C05374=1023.242,179.277,-116.475,168.477,48.773,159.154
C05375=1023.248,179.526,-116.498,168.481,48.767,159.153
C05376=1023.253,179.776,-116.521,168.485,48.762,159.153
C05377=1023.259,180.025,-116.544,168.489,48.757,159.152
C05378=1023.265,180.273,-116.565,168.492,48.752,159.151
C05379=1023.270,180.522,-116.588,168.496,48.746,159.151
C05380=1023.276,180.771,-116.611,168.501,48.741,159.151
C05381=1023.282,181.020,-116.632,168.504,48.735,159.150
C05382=1023.288,181.269,-116.655,168.508,48.730,159.149
C05383=1023.294,181.518,-116.678,168.511,48.725,159.149
C05384=1023.299,181.767,-116.701,168.516,48.719,159.148
C05385=1023.305,182.015,-116.723,168.519,48.714,159.148
C05386=1023.311,182.264,-116.745,168.523,48.708,159.147
C05387=1023.317,182.513,-116.768,168.526,48.703,159.147
C05388=1023.322,182.762,-116.791,168.531,48.698,159.146
C05389=1023.327,183.012,-116.814,168.534,48.693,159.146
C05390=1023.333,183.261,-116.837,168.537,48.688,159.145
C05391=1023.338,183.510,-116.861,168.541,48.683,159.145
C05392=1023.343,183.759,-116.884,168.545,48.678,159.144
C05393=1023.349,184.007,-116.906,168.549,48.673,159.144
C05394=1023.354,184.256,-116.930,168.553,48.668,159.143
C05395=1023.359,184.505,-116.953,168.556,48.662,159.143
C05396=1023.365,184.754,-116.976,168.560,48.657,159.142
C05397=1023.370,185.003,-117.000,168.564,48.652,159.142
C05398=1023.376,185.251,-117.023,168.568,48.647,159.141
C05399=1023.382,185.500,-117.046,168.571,48.642,159.141
C05400=1023.386,185.749,-117.069,168.575,48.637,159.140
C05401=1023.392,185.998,-117.092,168.579,48.632,159.140
C05402=1023.398,186.247,-117.115,168.582,48.627,159.139
C05403=1023.403,186.496,-117.138,168.587,48.622,159.139
C05404=1023.408,186.745,-117.161,168.590,48.616,159.138
C05405=1023.414,186.994,-117.184,168.594,48.611,159.138
C05406=1023.419,187.243,-117.208,168.598,48.606,159.137
C05407=1023.425,187.525,-117.234,168.603,48.600,159.137
C05408=1023.432,187.806,-117.261,168.607,48.594,159.136
C05409=1023.438,188.088,-117.287,168.611,48.589,159.136
C05410=1023.445,188.371,-117.313,168.615,48.583,159.135
C05411=1023.450,188.620,-117.337,168.619,48.578,159.135
C05412=1023.456,188.869,-117.360,168.623,48.573,159.134
C05413=1023.461,189.117,-117.383,168.627,48.568,159.134
C05414=1023.466,189.366,-117.406,168.631,48.563,159.133
C05415=1023.472,189.614,-117.430,168.635,48.558,159.133
C05416=1023.477,189.864,-117.453,168.638,48.552,159.132
C05417=1023.482,190.113,-117.476,168.643,48.547,159.132
C05418=1023.488,190.361,-117.499,168.646,48.542,159.131
C05419=1023.494,190.610,-117.524,168.651,48.537,159.131
C05420=1023.499,190.859,-117.547,168.654,48.532,159.130
C05421=1023.505,191.108,-117.570,168.658,48.527,159.130
C05422=1023.511,191.358,-117.593,168.662,48.521,159.129
C05423=1023.517,191.606,-117.617,168.666,48.517,159.129
C05424=1023.522,191.855,-117.640,168.670,48.512,159.128
C05425=1023.527,192.104,-117.664,168.674,48.507,159.128
C05426=1023.533,192.352,-117.687,168.678,48.502,159.127
C05427=1023.538,192.602,-117.711,168.681,48.496,159.127
C05428=1023.544,192.850,-117.734,168.686,48.491,159.126
C05429=1023.550,193.099,-117.757,168.690,48.486,159.126
C05430=1023.555,193.348,-117.781,168.694,48.481,159.125
C05431=1023.561,193.596,-117.805,168.698,48.476,159.125
C05432=1023.567,193.845,-117.828,168.701,48.471,159.125
C05433=1023.572,194.094,-117.851,168.706,48.465,159.124
C05434=1023.578,194.343,-117.875,168.710,48.460,159.124
C05435=1023.583,194.592,-117.898,168.713,48.456,159.123
C05436=1023.590,194.841,-117.922,168.718,48.450,159.123
C05437=1023.595,195.090,-117.945,168.721,48.446,159.122
C05438=1023.601,195.338,-117.970,168.726,48.440,159.122
C05439=1023.606,195.587,-117.992,168.730,48.435,159.121
C05440=1023.612,195.835,-118.016,168.733,48.430,159.121
C05441=1023.617,196.085,-118.040,168.738,48.425,159.120
C05442=1023.624,196.334,-118.064,168.742,48.420,159.120
C05443=1023.629,196.583,-118.087,168.746,48.415,159.119
C05444=1023.635,196.831,-118.111,168.750,48.410,159.119
C05445=1023.641,197.080,-118.134,168.754,48.405,159.119
C05446=1023.646,197.329,-118.158,168.758,48.400,159.118
C05447=1023.652,197.578,-118.181,168.762,48.395,159.118
C05448=1023.658,197.827,-118.206,168.766,48.389,159.117
C05449=1023.664,198.075,-118.229,168.770,48.384,159.117
C05450=1023.669,198.324,-118.252,168.774,48.379,159.116
C05451=1023.675,198.573,-118.277,168.779,48.374,159.116
C05452=1023.681,198.822,-118.300,168.782,48.369,159.115
C05453=1023.686,199.071,-118.324,168.787,48.364,159.115
C05454=1023.692,199.319,-118.348,168.791,48.359,159.114
C05455=1023.698,199.568,-118.371,168.795,48.354,159.114
C05456=1023.704,199.817,-118.395,168.799,48.349,159.113
C05457=1023.709,200.066,-118.420,168.803,48.344,159.113
C05458=1023.715,200.314,-118.443,168.807,48.339,159.113
C05459=1023.720,200.563,-118.467,168.811,48.334,159.112
C05460=1023.726,200.813,-118.491,168.816,48.329,159.112
C05461=1023.732,201.061,-118.516,168.819,48.324,159.111
C05462=1023.738,201.309,-118.539,168.824,48.319,159.111
C05463=1023.743,201.558,-118.564,168.828,48.314,159.110
C05464=1023.749,201.807,-118.588,168.832,48.309,159.110
C05465=1023.754,202.056,-118.612,168.836,48.304,159.109
C05466=1023.760,202.305,-118.635,168.841,48.300,159.109
C05467=1023.765,202.553,-118.660,168.844,48.295,159.109
C05468=1023.771,202.803,-118.684,168.849,48.290,159.108
C05469=1023.776,203.051,-118.709,168.853,48.285,159.108
C05470=1023.782,203.300,-118.732,168.857,48.280,159.107
C05471=1023.805,204.331,-118.833,169.270,48.380,159.187
C05472=1023.816,204.745,-118.876,169.275,48.373,159.186
C05473=1023.827,205.160,-118.919,169.281,48.366,159.186
C05474=1023.838,205.574,-118.961,169.286,48.359,159.185
C05475=1023.849,205.988,-119.004,169.292,48.352,159.184
C05476=1023.856,206.237,-119.031,169.295,48.349,159.184
C05477=1023.862,206.486,-119.056,169.298,48.344,159.184
C05478=1023.868,206.734,-119.082,169.301,48.341,159.183
C05479=1023.874,206.982,-119.108,169.305,48.336,159.183
C05480=1023.882,207.231,-119.134,169.307,48.333,159.182
C05481=1023.888,207.480,-119.159,169.311,48.329,159.182
C05482=1023.894,207.728,-119.185,169.314,48.325,159.182
C05483=1023.900,207.976,-119.211,169.318,48.321,159.181
C05484=1023.908,208.225,-119.237,169.320,48.317,159.181
C05485=1023.913,208.474,-119.263,169.324,48.313,159.180
C05486=1023.920,208.722,-119.289,169.327,48.309,159.180
C05487=1023.926,208.972,-119.315,169.331,48.305,159.180
C05488=1023.933,209.220,-119.341,169.333,48.301,159.179
C05489=1023.939,209.468,-119.367,169.337,48.297,159.179
C05490=1023.946,209.717,-119.393,169.340,48.293,159.179
C05491=1023.952,209.965,-119.419,169.344,48.289,159.178
C05492=1023.958,210.214,-119.445,169.346,48.285,159.178
C05493=1023.965,210.462,-119.471,169.350,48.282,159.178
C05494=1023.972,210.711,-119.497,169.353,48.278,159.177
C05495=1023.978,210.959,-119.524,169.356,48.274,159.177
C05496=1023.984,211.208,-119.549,169.360,48.270,159.176
C05497=1023.991,211.457,-119.575,169.362,48.266,159.176
C05498=1023.997,211.705,-119.602,169.366,48.263,159.176
C05499=1024.003,211.954,-119.627,169.369,48.259,159.175
C05500=1024.009,212.203,-119.654,169.373,48.255,159.175
C05501=1024.016,212.451,-119.681,169.376,48.251,159.175
C05502=1024.022,212.699,-119.707,169.379,48.247,159.174
C05503=1024.029,212.948,-119.734,169.382,48.244,159.174
C05504=1024.035,213.197,-119.759,169.386,48.240,159.174
C05505=1024.042,213.445,-119.785,169.389,48.236,159.173
C05506=1024.048,213.694,-119.812,169.393,48.232,159.173
C05507=1024.054,213.942,-119.838,169.396,48.229,159.173
C05508=1024.061,214.191,-119.865,169.399,48.225,159.172
C05509=1024.067,214.439,-119.890,169.402,48.221,159.172
C05510=1024.073,214.688,-119.916,169.406,48.217,159.172
C05511=1024.080,214.937,-119.943,169.409,48.214,159.171
C05512=1024.086,215.185,-119.970,169.412,48.210,159.171
C05513=1024.093,215.433,-119.996,169.415,48.206,159.171
C05514=1024.099,215.682,-120.023,169.418,48.202,159.170
C05515=1024.106,215.930,-120.049,169.422,48.198,159.170
C05516=1024.112,216.179,-120.076,169.425,48.195,159.170
C05517=1024.119,216.427,-120.102,169.429,48.191,159.169
C05518=1024.125,216.676,-120.127,169.432,48.187,159.169
C05519=1024.131,216.925,-120.154,169.435,48.183,159.169
C05520=1024.138,217.173,-120.181,169.439,48.180,159.168
C05521=1024.145,217.421,-120.207,169.442,48.176,159.168
C05522=1024.151,217.670,-120.234,169.445,48.172,159.168
C05523=1024.158,217.919,-120.260,169.449,48.169,159.167
C05524=1024.164,218.168,-120.287,169.452,48.165,159.167
C05525=1024.171,218.416,-120.313,169.456,48.161,159.167
C05526=1024.178,218.664,-120.339,169.459,48.158,159.166
C05527=1024.183,218.913,-120.366,169.462,48.154,159.166
C05528=1024.194,219.329,-120.410,169.468,48.148,159.165
C05529=1024.205,219.746,-120.456,169.474,48.142,159.165
C05530=1024.215,220.162,-120.500,169.479,48.136,159.165
C05531=1024.227,220.579,-120.545,169.485,48.130,159.164
C05532=1024.232,220.828,-120.572,169.488,48.127,159.164
C05533=1024.239,221.077,-120.599,169.491,48.123,159.163
C05534=1024.245,221.325,-120.625,169.495,48.120,159.163
C05535=1024.252,221.574,-120.652,169.498,48.116,159.163
C05536=1024.258,221.822,-120.679,169.502,48.112,159.163
C05537=1024.265,222.070,-120.706,169.505,48.109,159.162
C05538=1024.271,222.319,-120.732,169.509,48.105,159.162
C05539=1024.277,222.568,-120.759,169.512,48.102,159.162
C05540=1024.284,222.815,-120.786,169.516,48.098,159.161
C05541=1024.290,223.064,-120.813,169.519,48.095,159.161
C05542=1024.297,223.313,-120.840,169.521,48.091,159.161
C05543=1024.303,223.561,-120.866,169.525,48.088,159.161
C05544=1024.310,223.810,-120.894,169.529,48.085,159.160
C05545=1024.316,224.058,-120.921,169.532,48.080,159.160
C05546=1024.323,224.307,-120.947,169.535,48.077,159.160
C05547=1024.329,224.555,-120.975,169.539,48.074,159.160
C05548=1024.335,224.804,-121.002,169.542,48.070,159.159
C05549=1024.342,225.053,-121.028,169.546,48.067,159.159
C05550=1024.348,225.300,-121.055,169.549,48.064,159.159
C05551=1024.355,225.549,-121.082,169.553,48.060,159.158
C05552=1024.361,225.797,-121.108,169.556,48.056,159.158
C05553=1024.368,226.046,-121.136,169.560,48.053,159.158
C05554=1024.374,226.295,-121.163,169.563,48.049,159.158
C05555=1024.380,226.543,-121.190,169.567,48.046,159.157
C05556=1024.388,226.791,-121.217,169.570,48.043,159.157
C05557=1024.394,227.040,-121.244,169.573,48.039,159.157
C05558=1024.400,227.288,-121.271,169.577,48.035,159.157
C05559=1024.406,227.537,-121.298,169.580,48.032,159.156
C05560=1024.412,227.785,-121.326,169.584,48.029,159.156
C05561=1024.420,228.034,-121.352,169.587,48.026,159.156
C05562=1024.426,228.282,-121.380,169.591,48.022,159.156
C05563=1024.432,228.531,-121.406,169.594,48.019,159.155
C05564=1024.439,228.779,-121.434,169.598,48.015,159.155
C05565=1024.445,229.028,-121.461,169.601,48.012,159.155
C05566=1024.451,229.276,-121.489,169.604,48.009,159.155
C05567=1024.458,229.524,-121.516,169.608,48.006,159.154
C05568=1024.464,229.773,-121.543,169.611,48.003,159.154
C05569=1024.470,230.021,-121.571,169.616,47.999,159.154
C05570=1024.477,230.269,-121.598,169.618,47.995,159.154
C05571=1024.483,230.519,-121.625,169.622,47.992,159.153
C05572=1024.490,230.767,-121.653,169.625,47.989,159.153
C05573=1024.496,231.015,-121.681,169.629,47.986,159.153
C05574=1024.502,231.264,-121.708,169.633,47.982,159.153
C05575=1024.509,231.512,-121.735,169.636,47.979,159.153
C05576=1024.515,231.760,-121.763,169.640,47.976,159.152
C05577=1024.522,232.009,-121.790,169.643,47.973,159.152
C05578=1024.528,232.257,-121.817,169.647,47.969,159.152
C05579=1024.534,232.505,-121.845,169.650,47.966,159.152
C05580=1024.541,232.754,-121.872,169.653,47.963,159.151
C05581=1024.548,233.002,-121.900,169.657,47.960,159.151
C05582=1024.553,233.251,-121.928,169.660,47.957,159.151
C05583=1024.559,233.499,-121.955,169.664,47.953,159.151
C05584=1024.570,233.908,-122.000,169.670,47.949,159.151
C05585=1024.581,234.317,-122.045,169.676,47.943,159.150
C05586=1024.591,234.726,-122.092,169.682,47.938,159.150
C05587=1024.602,235.134,-122.137,169.688,47.932,159.150
C05588=1024.609,235.383,-122.165,169.691,47.929,159.149
C05589=1024.615,235.631,-122.192,169.695,47.926,159.149
C05590=1024.622,235.880,-122.219,169.698,47.923,159.149
C05591=1024.628,236.129,-122.247,169.702,47.919,159.149
C05592=1024.634,236.377,-122.274,169.705,47.917,159.149
C05593=1024.641,236.625,-122.302,169.709,47.914,159.148
C05594=1024.647,236.874,-122.331,169.712,47.910,159.148
C05595=1024.654,237.122,-122.358,169.717,47.907,159.148
C05596=1024.660,237.371,-122.386,169.720,47.904,159.148
C05597=1024.667,237.619,-122.414,169.723,47.901,159.147
C05598=1024.673,237.867,-122.441,169.727,47.898,159.148
C05599=1024.680,238.115,-122.469,169.730,47.895,159.147
C05600=1024.686,238.364,-122.497,169.734,47.892,159.147
C05601=1024.693,238.612,-122.525,169.737,47.888,159.147
C05602=1024.699,238.861,-122.553,169.741,47.885,159.147
C05603=1024.706,239.109,-122.580,169.745,47.883,159.147
C05604=1024.713,239.358,-122.608,169.749,47.879,159.146
C05605=1024.719,239.606,-122.636,169.752,47.876,159.146
C05606=1024.725,239.854,-122.664,169.755,47.873,159.146
C05607=1024.732,240.102,-122.692,169.759,47.870,159.146
C05608=1024.738,240.351,-122.720,169.763,47.867,159.146
C05609=1024.744,240.599,-122.748,169.767,47.864,159.145
C05610=1024.751,240.848,-122.776,169.770,47.861,159.145
C05611=1024.757,241.096,-122.805,169.774,47.858,159.145
C05612=1024.764,241.344,-122.833,169.777,47.855,159.145
C05613=1024.770,241.593,-122.861,169.781,47.852,159.145
C05614=1024.776,241.841,-122.888,169.785,47.849,159.145
C05615=1024.783,242.089,-122.917,169.788,47.847,159.145
C05616=1024.789,242.337,-122.945,169.792,47.843,159.144
C05617=1024.795,242.586,-122.973,169.795,47.840,159.144
C05618=1024.802,242.834,-123.002,169.800,47.837,159.144
C05619=1024.808,243.082,-123.030,169.803,47.834,159.144
C05620=1024.814,243.331,-123.058,169.806,47.832,159.144
C05621=1024.821,243.579,-123.086,169.810,47.829,159.144
C05622=1024.828,243.827,-123.114,169.814,47.826,159.144
C05623=1024.834,244.076,-123.143,169.818,47.823,159.143
C05624=1024.840,244.324,-123.172,169.821,47.820,159.143
C05625=1024.847,244.573,-123.199,169.824,47.817,159.143
C05626=1024.853,244.821,-123.228,169.829,47.814,159.143
C05627=1024.859,245.070,-123.257,169.832,47.812,159.143
C05628=1024.865,245.317,-123.285,169.836,47.809,159.143
C05629=1024.871,245.565,-123.313,169.840,47.806,159.143
C05630=1024.878,245.814,-123.342,169.843,47.803,159.143
C05631=1024.884,246.062,-123.371,169.847,47.800,159.143
C05632=1024.891,246.310,-123.399,169.850,47.798,159.143
C05633=1024.897,246.558,-123.428,169.855,47.795,159.142
C05634=1024.903,246.807,-123.456,169.858,47.792,159.142
C05635=1024.909,247.055,-123.485,169.861,47.790,159.142
C05636=1024.916,247.304,-123.513,169.865,47.786,159.142
C05637=1024.922,247.552,-123.542,169.869,47.784,159.142
C05638=1024.928,247.800,-123.571,169.873,47.781,159.142
C05639=1024.935,248.048,-123.599,169.876,47.778,159.142
C05640=1024.945,248.451,-123.645,169.882,47.773,159.141
C05641=1024.955,248.854,-123.693,169.888,47.769,159.141
C05642=1024.966,249.256,-123.739,169.895,47.765,159.141
C05643=1024.976,249.660,-123.785,169.901,47.760,159.141
C05644=1024.983,249.908,-123.814,169.904,47.758,159.141
C05645=1024.990,250.156,-123.843,169.909,47.755,159.141
C05646=1024.996,250.404,-123.872,169.912,47.752,159.141
C05647=1025.002,250.652,-123.900,169.916,47.749,159.141
C05648=1025.009,250.900,-123.928,169.920,47.747,159.141
C05649=1025.015,251.148,-123.958,169.923,47.744,159.141
C05650=1025.021,251.397,-123.987,169.927,47.741,159.141
C05651=1025.027,251.645,-124.015,169.931,47.738,159.140
C05652=1025.035,251.894,-124.044,169.935,47.736,159.140
C05653=1025.041,252.142,-124.073,169.938,47.733,159.140
C05654=1025.047,252.390,-124.102,169.943,47.731,159.140
C05655=1025.053,252.638,-124.131,169.946,47.728,159.140
C05656=1025.060,252.887,-124.159,169.950,47.725,159.140
C05657=1025.066,253.135,-124.188,169.954,47.722,159.140
C05658=1025.073,253.383,-124.217,169.958,47.720,159.140
C05659=1025.080,253.631,-124.245,169.962,47.717,159.140
C05660=1025.086,253.880,-124.274,169.965,47.715,159.140
C05661=1025.093,254.128,-124.304,169.969,47.712,159.140
C05662=1025.099,254.376,-124.333,169.972,47.709,159.139
C05663=1025.106,254.624,-124.361,169.977,47.706,159.139
C05664=1025.113,254.872,-124.390,169.980,47.704,159.139
C05665=1025.119,255.121,-124.419,169.985,47.701,159.139
C05666=1025.125,255.369,-124.448,169.988,47.699,159.139
C05667=1025.132,255.617,-124.476,169.992,47.696,159.139
C05668=1025.139,255.866,-124.506,169.996,47.693,159.139
C05669=1025.145,256.114,-124.535,170.000,47.691,159.139
C05670=1025.151,256.362,-124.564,170.003,47.688,159.139
C05671=1025.158,256.610,-124.592,170.008,47.685,159.139
C05672=1025.165,256.859,-124.622,170.011,47.683,159.139
C05673=1025.171,257.107,-124.651,170.016,47.680,159.139
C05674=1025.178,257.355,-124.680,170.019,47.677,159.139
C05675=1025.186,257.603,-124.709,170.023,47.675,159.139
C05676=1025.192,257.851,-124.738,170.027,47.672,159.139
C05677=1025.198,258.099,-124.767,170.031,47.670,159.139
C05678=1025.204,258.347,-124.796,170.035,47.667,159.139
C05679=1025.212,258.596,-124.825,170.039,47.664,159.139
C05680=1025.218,258.844,-124.854,170.043,47.662,159.139
C05681=1025.224,259.092,-124.883,170.047,47.659,159.139
C05682=1025.231,259.341,-124.913,170.050,47.657,159.138
C05683=1025.238,259.589,-124.941,170.055,47.654,159.138
C05684=1025.245,259.838,-124.970,170.058,47.652,159.138
C05685=1025.252,260.085,-125.000,170.063,47.649,159.138
C05686=1025.258,260.333,-125.029,170.066,47.647,159.138
C05687=1025.266,260.582,-125.058,170.070,47.644,159.138
C05688=1025.272,260.830,-125.087,170.074,47.641,159.138
C05689=1025.278,261.078,-125.117,170.079,47.639,159.138
C05690=1025.284,261.327,-125.147,170.082,47.637,159.138
C05691=1025.291,261.575,-125.176,170.086,47.634,159.138
C05692=1025.297,261.822,-125.206,170.090,47.632,159.138
C05693=1025.304,262.071,-125.235,170.094,47.629,159.138
C05694=1025.311,262.319,-125.265,170.098,47.627,159.138
C05695=1025.317,262.567,-125.294,170.102,47.625,159.138
C05696=1025.327,262.968,-125.343,170.108,47.621,159.138
C05697=1025.338,263.369,-125.390,170.115,47.617,159.138
C05698=1025.348,263.771,-125.438,170.121,47.614,159.138
C05699=1025.359,264.172,-125.486,170.128,47.609,159.138
C05700=1025.365,264.420,-125.516,170.132,47.607,159.138
C05701=1025.372,264.668,-125.545,170.136,47.605,159.138
C05702=1025.379,264.916,-125.575,170.140,47.602,159.138
C05703=1025.384,265.164,-125.604,170.143,47.600,159.138
C05704=1025.391,265.413,-125.634,170.148,47.598,159.138
C05705=1025.398,265.660,-125.664,170.151,47.596,159.138
C05706=1025.405,265.909,-125.694,170.156,47.593,159.138
C05707=1025.411,266.156,-125.723,170.159,47.591,159.138
C05708=1025.418,266.405,-125.754,170.164,47.588,159.138
C05709=1025.424,266.653,-125.783,170.168,47.587,159.139
C05710=1025.431,266.901,-125.813,170.172,47.584,159.139
C05711=1025.437,267.149,-125.844,170.176,47.582,159.139
C05712=1025.444,267.398,-125.873,170.180,47.579,159.139
C05713=1025.450,267.645,-125.903,170.184,47.578,159.139
C05714=1025.458,267.894,-125.933,170.188,47.575,159.139
C05715=1025.463,268.141,-125.963,170.192,47.573,159.139
C05716=1025.470,268.390,-125.993,170.196,47.571,159.139
C05717=1025.476,268.638,-126.023,170.200,47.569,159.139
C05718=1025.483,268.886,-126.053,170.205,47.566,159.139
C05719=1025.490,269.134,-126.083,170.208,47.564,159.139
C05720=1025.496,269.382,-126.114,170.213,47.562,159.139
C05721=1025.503,269.630,-126.143,170.216,47.560,159.139
C05722=1025.510,269.879,-126.173,170.221,47.557,159.139
C05723=1025.515,270.126,-126.203,170.225,47.555,159.139
C05724=1025.523,270.375,-126.233,170.229,47.553,159.139
C05725=1025.528,270.623,-126.264,170.233,47.551,159.139
C05726=1025.536,270.871,-126.294,170.237,47.549,159.139
C05727=1025.541,271.119,-126.324,170.241,47.546,159.139
C05728=1025.549,271.367,-126.354,170.246,47.544,159.140
C05729=1025.555,271.615,-126.385,170.249,47.543,159.140
C05730=1025.562,271.863,-126.415,170.254,47.540,159.140
C05731=1025.568,272.111,-126.445,170.257,47.538,159.140
C05732=1025.575,272.359,-126.475,170.262,47.536,159.140
C05733=1025.581,272.607,-126.506,170.266,47.534,159.140
C05734=1025.588,272.856,-126.536,170.270,47.532,159.140
C05735=1025.594,273.103,-126.566,170.274,47.530,159.140
C05736=1025.601,273.352,-126.596,170.279,47.528,159.140
C05737=1025.607,273.599,-126.628,170.282,47.526,159.140
C05738=1025.614,273.847,-126.658,170.287,47.523,159.140
C05739=1025.621,274.096,-126.688,170.292,47.521,159.140
C05740=1025.627,274.343,-126.718,170.295,47.520,159.141
C05741=1025.634,274.592,-126.749,170.300,47.517,159.141
C05742=1025.640,274.840,-126.780,170.304,47.516,159.141
C05743=1025.647,275.087,-126.810,170.308,47.513,159.141
C05744=1025.653,275.336,-126.841,170.312,47.511,159.141
C05745=1025.661,275.584,-126.871,170.317,47.509,159.141
C05746=1025.666,275.832,-126.901,170.320,47.507,159.141
C05747=1025.673,276.079,-126.933,170.325,47.505,159.141
C05748=1025.680,276.328,-126.963,170.329,47.504,159.141
C05749=1025.687,276.576,-126.993,170.333,47.501,159.141
C05750=1025.693,276.824,-127.023,170.337,47.499,159.142
C05751=1025.700,277.072,-127.055,170.342,47.497,159.142
C05752=1025.711,277.478,-127.105,170.348,47.494,159.142
C05753=1025.721,277.883,-127.155,170.356,47.491,159.142
C05754=1025.732,278.289,-127.205,170.362,47.488,159.142
C05755=1025.743,278.695,-127.257,170.370,47.485,159.143
C05756=1025.749,278.943,-127.287,170.374,47.483,159.143
C05757=1025.756,279.190,-127.318,170.379,47.481,159.143
C05758=1025.762,279.439,-127.348,170.382,47.479,159.143
C05759=1025.769,279.687,-127.380,170.387,47.477,159.143
C05760=1025.776,279.935,-127.411,170.391,47.475,159.143
C05761=1025.782,280.182,-127.442,170.395,47.473,159.143
C05762=1025.788,280.431,-127.472,170.399,47.472,159.144
C05763=1025.795,280.679,-127.504,170.404,47.470,159.144
C05764=1025.802,280.926,-127.535,170.408,47.468,159.144
C05765=1025.809,281.175,-127.565,170.413,47.466,159.144
C05766=1025.815,281.422,-127.596,170.417,47.464,159.144
C05767=1025.821,281.671,-127.627,170.421,47.463,159.144
C05768=1025.828,281.919,-127.659,170.426,47.461,159.145
C05769=1025.835,282.167,-127.690,170.430,47.459,159.145
C05770=1025.842,282.415,-127.720,170.434,47.457,159.145
C05771=1025.849,282.663,-127.752,170.438,47.455,159.145
C05772=1025.855,282.911,-127.783,170.443,47.454,159.145
C05773=1025.861,283.158,-127.814,170.448,47.452,159.145
C05774=1025.868,283.406,-127.845,170.452,47.450,159.146
C05775=1025.875,283.654,-127.876,170.456,47.448,159.146
C05776=1025.881,283.902,-127.908,170.460,47.447,159.146
C05777=1025.889,284.150,-127.938,170.465,47.445,159.146
C05778=1025.895,284.398,-127.969,170.469,47.443,159.146
C05779=1025.902,284.646,-128.001,170.474,47.441,159.146
C05780=1025.909,284.894,-128.032,170.478,47.439,159.147
C05781=1025.915,285.142,-128.064,170.482,47.438,159.147
C05782=1025.922,285.390,-128.095,170.487,47.436,159.147
C05783=1025.929,285.638,-128.126,170.491,47.434,159.147
C05784=1025.935,285.886,-128.157,170.496,47.432,159.147
C05785=1025.941,286.133,-128.188,170.501,47.430,159.148
C05786=1025.948,286.381,-128.220,170.505,47.429,159.148
C05787=1025.955,286.629,-128.251,170.509,47.427,159.148
C05788=1025.962,286.877,-128.282,170.513,47.426,159.148
C05789=1025.968,287.125,-128.314,170.518,47.424,159.148
C05790=1025.975,287.373,-128.345,170.523,47.422,159.149
C05791=1025.982,287.621,-128.377,170.527,47.421,159.149
C05792=1025.989,287.868,-128.409,170.532,47.419,159.149
C05793=1025.995,288.116,-128.440,170.536,47.418,159.149
C05794=1026.001,288.364,-128.472,170.540,47.416,159.150
C05795=1026.008,288.612,-128.504,170.545,47.414,159.150
C05796=1026.015,288.860,-128.535,170.549,47.413,159.150
C05797=1026.022,289.108,-128.567,170.554,47.411,159.150
C05798=1026.028,289.356,-128.598,170.558,47.409,159.150
C05799=1026.035,289.603,-128.630,170.563,47.408,159.151
C05800=1026.043,289.852,-128.662,170.568,47.406,159.151
C05801=1026.049,290.100,-128.694,170.572,47.405,159.151
C05802=1026.055,290.348,-128.725,170.576,47.403,159.151
C05803=1026.062,290.596,-128.757,170.581,47.401,159.152
C05804=1026.069,290.843,-128.789,170.586,47.400,159.152
C05805=1026.076,291.091,-128.821,170.590,47.398,159.152
C05806=1026.082,291.339,-128.853,170.594,47.397,159.152
C05807=1026.089,291.586,-128.885,170.599,47.395,159.153
C05808=1026.101,292.005,-128.938,170.607,47.393,159.153
C05809=1026.112,292.423,-128.992,170.615,47.390,159.153
C05810=1026.123,292.840,-129.046,170.623,47.388,159.154
C05811=1026.134,293.259,-129.099,170.630,47.385,159.154
C05812=1026.141,293.506,-129.131,170.635,47.384,159.155
C05813=1026.148,293.755,-129.164,170.640,47.382,159.155
C05814=1026.155,294.002,-129.196,170.644,47.381,159.155
C05815=1026.161,294.250,-129.228,170.649,47.379,159.155
C05816=1026.168,294.498,-129.260,170.654,47.378,159.156
C05817=1026.174,294.745,-129.293,170.658,47.377,159.156
C05818=1026.180,294.993,-129.325,170.663,47.375,159.156
C05819=1026.187,295.241,-129.357,170.667,47.374,159.157
C05820=1026.194,295.489,-129.390,170.672,47.373,159.157
C05821=1026.201,295.736,-129.422,170.677,47.371,159.157
C05822=1026.207,295.985,-129.454,170.681,47.370,159.158
C05823=1026.213,296.232,-129.487,170.686,47.369,159.158
C05824=1026.221,296.479,-129.519,170.690,47.368,159.158
C05825=1026.227,296.728,-129.552,170.695,47.366,159.158
C05826=1026.233,296.976,-129.584,170.700,47.365,159.159
C05827=1026.240,297.223,-129.616,170.704,47.364,159.159
C05828=1026.247,297.471,-129.649,170.709,47.362,159.159
C05829=1026.253,297.718,-129.682,170.714,47.361,159.160
C05830=1026.261,297.966,-129.714,170.718,47.360,159.160
C05831=1026.267,298.215,-129.746,170.723,47.358,159.160
C05832=1026.273,298.462,-129.779,170.728,47.357,159.161
C05833=1026.280,298.709,-129.811,170.732,47.356,159.161
C05834=1026.287,298.958,-129.844,170.737,47.355,159.161
C05835=1026.294,299.205,-129.876,170.742,47.353,159.162
C05836=1026.300,299.453,-129.909,170.747,47.353,159.162
C05837=1026.307,299.701,-129.942,170.752,47.351,159.162
C05838=1026.314,299.948,-129.974,170.757,47.350,159.163
C05839=1026.320,300.196,-130.007,170.761,47.349,159.163
C05840=1026.327,300.444,-130.040,170.766,47.347,159.163
C05841=1026.334,300.691,-130.072,170.771,47.346,159.164
C05842=1026.341,300.939,-130.105,170.775,47.345,159.164
C05843=1026.347,301.187,-130.138,170.780,47.344,159.165
C05844=1026.355,301.435,-130.170,170.785,47.343,159.165
C05845=1026.361,301.683,-130.204,170.790,47.341,159.165
C05846=1026.368,301.930,-130.236,170.794,47.340,159.165
C05847=1026.375,302.178,-130.268,170.799,47.339,159.166
C05848=1026.382,302.426,-130.302,170.805,47.338,159.166
C05849=1026.388,302.673,-130.335,170.810,47.337,159.167
C05850=1026.396,302.921,-130.368,170.814,47.335,159.167
C05851=1026.402,303.169,-130.400,170.819,47.334,159.167
C05852=1026.408,303.416,-130.433,170.824,47.333,159.168
C05853=1026.416,303.664,-130.466,170.828,47.332,159.168
C05854=1026.422,303.912,-130.498,170.833,47.331,159.168
C05855=1026.430,304.159,-130.532,170.839,47.330,159.169
C05856=1026.437,304.407,-130.564,170.844,47.329,159.169
C05857=1026.444,304.655,-130.597,170.848,47.328,159.169
C05858=1026.450,304.903,-130.630,170.853,47.327,159.170
C05859=1026.458,305.150,-130.663,170.858,47.325,159.170
C05860=1026.464,305.397,-130.696,170.863,47.324,159.171
C05861=1026.471,305.646,-130.729,170.869,47.323,159.171
C05862=1026.479,305.893,-130.762,170.873,47.322,159.171
C05863=1026.485,306.141,-130.795,170.878,47.321,159.172
C05864=1026.491,306.358,-130.824,170.882,47.320,159.172
C05865=1026.497,306.576,-130.853,170.887,47.319,159.173
C05866=1026.504,306.794,-130.882,170.891,47.318,159.173
C05867=1026.510,307.012,-130.911,170.895,47.317,159.173
C05868=1026.516,307.228,-130.941,170.899,47.316,159.174
C05869=1026.522,307.446,-130.970,170.904,47.316,159.174
C05870=1026.529,307.664,-130.999,170.909,47.314,159.174
C05871=1026.534,307.882,-131.028,170.913,47.313,159.175
C05872=1026.542,308.130,-131.060,170.918,47.312,159.175
C05873=1026.548,308.377,-131.094,170.923,47.311,159.175
C05874=1026.555,308.625,-131.127,170.928,47.310,159.176
C05875=1026.563,308.873,-131.160,170.933,47.309,159.176
C05876=1026.570,309.120,-131.194,170.938,47.308,159.177
C05877=1026.577,309.368,-131.227,170.943,47.307,159.177
C05878=1026.584,309.616,-131.261,170.948,47.306,159.178
C05879=1026.591,309.863,-131.293,170.954,47.305,159.178
C05880=1026.598,310.110,-131.327,170.958,47.304,159.178
C05881=1026.605,310.358,-131.360,170.963,47.303,159.179
C05882=1026.612,310.605,-131.393,170.968,47.302,159.179
C05883=1026.620,310.853,-131.426,170.973,47.301,159.180
C05884=1026.626,311.101,-131.461,170.979,47.300,159.180
C05885=1026.633,311.348,-131.494,170.983,47.300,159.181
C05886=1026.640,311.596,-131.528,170.989,47.299,159.181
C05887=1026.647,311.843,-131.562,170.994,47.298,159.182
C05888=1026.653,312.091,-131.596,170.999,47.297,159.182
C05889=1026.660,312.338,-131.630,171.004,47.296,159.183
C05890=1026.667,312.586,-131.664,171.009,47.296,159.183
C05891=1026.674,312.834,-131.698,171.014,47.295,159.184
C05892=1026.680,313.081,-131.732,171.019,47.294,159.184
C05893=1026.688,313.329,-131.765,171.025,47.293,159.185
C05894=1026.694,313.577,-131.800,171.030,47.293,159.185
C05895=1026.701,313.824,-131.833,171.034,47.292,159.186
C05896=1026.708,314.071,-131.867,171.040,47.291,159.186
C05897=1026.714,314.319,-131.901,171.045,47.291,159.187
C05898=1026.721,314.567,-131.935,171.050,47.290,159.187
C05899=1026.729,314.815,-131.969,171.056,47.289,159.188
C05900=1026.735,315.062,-132.003,171.061,47.288,159.188
C05901=1026.742,315.309,-132.038,171.065,47.288,159.189
C05902=1026.749,315.557,-132.072,171.071,47.287,159.189
C05903=1026.756,315.805,-132.106,171.076,47.286,159.190
C05904=1026.763,316.052,-132.140,171.082,47.286,159.190
C05905=1026.770,316.300,-132.174,171.087,47.285,159.191
C05906=1026.776,316.547,-132.208,171.092,47.284,159.191
C05907=1026.783,316.794,-132.242,171.098,47.283,159.192
C05908=1026.791,317.042,-132.276,171.102,47.283,159.192
C05909=1026.797,317.290,-132.310,171.108,47.283,159.193
C05910=1026.805,317.537,-132.345,171.113,47.282,159.193
C05911=1026.812,317.785,-132.379,171.118,47.281,159.194
C05912=1026.818,318.033,-132.413,171.124,47.280,159.194
C05913=1026.826,318.280,-132.448,171.129,47.280,159.195
C05914=1026.833,318.527,-132.482,171.134,47.279,159.195
C05915=1026.840,318.775,-132.517,171.140,47.279,159.196
C05916=1026.847,319.022,-132.551,171.145,47.278,159.197
C05917=1026.854,319.270,-132.584,171.150,47.277,159.197
C05918=1026.861,319.517,-132.619,171.155,47.277,159.198
C05919=1026.868,319.765,-132.653,171.161,47.276,159.198
C05920=1026.876,320.012,-132.688,171.166,47.276,159.199
C05921=1026.882,320.260,-132.722,171.171,47.275,159.199
C05922=1026.890,320.507,-132.757,171.177,47.274,159.200
C05923=1026.897,320.755,-132.791,171.182,47.274,159.200
C05924=1026.903,320.975,-132.822,171.187,47.273,159.201
C05925=1026.909,321.196,-132.853,171.192,47.273,159.201
C05926=1026.915,321.415,-132.884,171.196,47.272,159.202
C05927=1026.922,321.636,-132.914,171.202,47.272,159.203
C05928=1026.928,321.856,-132.945,171.206,47.272,159.203
C05929=1026.935,322.076,-132.976,171.212,47.271,159.203
C05930=1026.941,322.296,-133.006,171.216,47.270,159.204
C05931=1026.948,322.516,-133.037,171.220,47.270,159.204
C05932=1026.955,322.763,-133.071,171.226,47.270,159.205
C05933=1026.962,323.011,-133.106,171.231,47.269,159.206
C05934=1026.970,323.258,-133.141,171.237,47.269,159.206
C05935=1026.977,323.506,-133.175,171.242,47.268,159.207
C05936=1026.984,323.754,-133.210,171.248,47.268,159.207
C05937=1026.991,324.001,-133.244,171.253,47.267,159.208
C05938=1026.999,324.248,-133.279,171.259,47.267,159.209
C05939=1027.006,324.496,-133.314,171.265,47.266,159.209
C05940=1027.013,324.743,-133.348,171.270,47.266,159.210
C05941=1027.020,324.991,-133.383,171.276,47.265,159.210
C05942=1027.028,325.239,-133.418,171.281,47.265,159.211
C05943=1027.036,325.486,-133.453,171.287,47.264,159.212
C05944=1027.042,325.733,-133.488,171.293,47.264,159.212
C05945=1027.050,325.981,-133.522,171.299,47.263,159.213
C05946=1027.057,326.229,-133.557,171.304,47.263,159.214
C05947=1027.064,326.476,-133.592,171.310,47.263,159.214
C05948=1027.073,326.723,-133.627,171.315,47.262,159.215
C05949=1027.079,326.971,-133.662,171.321,47.262,159.215
C05950=1027.087,327.218,-133.696,171.327,47.262,159.216
C05951=1027.094,327.466,-133.732,171.332,47.261,159.217
C05952=1027.102,327.713,-133.766,171.338,47.261,159.217
C05953=1027.109,327.960,-133.802,171.343,47.261,159.218
C05954=1027.116,328.208,-133.838,171.349,47.260,159.219
C05955=1027.123,328.455,-133.873,171.355,47.260,159.219
C05956=1027.130,328.703,-133.908,171.360,47.259,159.220
C05957=1027.138,328.950,-133.944,171.366,47.259,159.221
C05958=1027.145,329.197,-133.979,171.371,47.259,159.221
C05959=1027.152,329.444,-134.014,171.377,47.259,159.222
C05960=1027.159,329.692,-134.050,171.382,47.259,159.223
C05961=1027.166,329.939,-134.085,171.388,47.259,159.223
C05962=1027.173,330.187,-134.121,171.394,47.259,159.224
C05963=1027.181,330.434,-134.156,171.400,47.258,159.225
C05964=1027.188,330.681,-134.191,171.406,47.258,159.226
C05965=1027.195,330.929,-134.227,171.412,47.258,159.226
C05966=1027.202,331.176,-134.263,171.417,47.258,159.227
C05967=1027.210,331.424,-134.298,171.423,47.257,159.228
C05968=1027.217,331.671,-134.334,171.429,47.257,159.228
C05969=1027.225,331.918,-134.369,171.434,47.257,159.229
C05970=1027.232,332.165,-134.405,171.440,47.257,159.230
C05971=1027.239,332.413,-134.440,171.446,47.257,159.230
C05972=1027.247,332.660,-134.476,171.451,47.257,159.231
C05973=1027.254,332.908,-134.512,171.458,47.256,159.232
C05974=1027.262,333.156,-134.548,171.464,47.257,159.233
C05975=1027.269,333.402,-134.583,171.470,47.257,159.233
C05976=1027.277,333.650,-134.619,171.475,47.256,159.234
C05977=1027.284,333.897,-134.654,171.481,47.256,159.235
C05978=1027.292,334.144,-134.691,171.487,47.256,159.236
C05979=1027.298,334.392,-134.726,171.493,47.256,159.236
C05980=1027.306,334.639,-134.762,171.499,47.256,159.237
C05981=1027.313,334.887,-134.799,171.505,47.256,159.238
C05982=1027.320,335.134,-134.835,171.511,47.256,159.239
C05983=1027.328,335.381,-134.871,171.517,47.256,159.239
C05984=1027.334,335.598,-134.902,171.521,47.256,159.240
C05985=1027.340,335.817,-134.934,171.527,47.256,159.241
C05986=1027.348,336.035,-134.966,171.533,47.256,159.241
C05987=1027.354,336.252,-134.997,171.537,47.256,159.242
C05988=1027.360,336.470,-135.029,171.543,47.256,159.243
C05989=1027.367,336.688,-135.061,171.548,47.257,159.244
C05990=1027.373,336.906,-135.093,171.553,47.256,159.244
C05991=1027.380,337.124,-135.125,171.558,47.257,159.245
C05992=1027.387,337.372,-135.161,171.565,47.256,159.246
C05993=1027.394,337.618,-135.197,171.571,47.257,159.247
C05994=1027.402,337.866,-135.233,171.576,47.256,159.247
C05995=1027.410,338.113,-135.269,171.582,47.257,159.248
C05996=1027.417,338.361,-135.306,171.588,47.257,159.249
C05997=1027.424,338.608,-135.342,171.595,47.257,159.250
C05998=1027.432,338.855,-135.378,171.601,47.257,159.250
C05999=1027.439,339.102,-135.415,171.607,47.257,159.251
C06000=1027.447,339.349,-135.451,171.613,47.258,159.252
C06001=1027.455,339.597,-135.488,171.619,47.257,159.253
C06002=1027.462,339.844,-135.523,171.625,47.258,159.254
C06003=1027.470,340.091,-135.560,171.631,47.258,159.255
C06004=1027.478,340.338,-135.597,171.637,47.258,159.255
C06005=1027.485,340.586,-135.633,171.644,47.258,159.256
C06006=1027.492,340.833,-135.670,171.650,47.258,159.257
C06007=1027.500,341.080,-135.707,171.655,47.258,159.258
C06008=1027.507,341.328,-135.743,171.661,47.259,159.259
C06009=1027.514,341.574,-135.780,171.668,47.259,159.260
C06010=1027.522,341.821,-135.816,171.674,47.259,159.261
C06011=1027.529,342.068,-135.854,171.680,47.260,159.261
C06012=1027.537,342.316,-135.890,171.686,47.260,159.262
C06013=1027.544,342.563,-135.927,171.693,47.260,159.263
C06014=1027.552,342.810,-135.964,171.699,47.260,159.264
C06015=1027.560,343.057,-136.001,171.705,47.261,159.265
C06016=1027.567,343.305,-136.037,171.712,47.261,159.266
C06017=1027.575,343.552,-136.074,171.718,47.261,159.267
C06018=1027.583,343.799,-136.111,171.724,47.262,159.268
C06019=1027.590,344.046,-136.148,171.731,47.262,159.268
C06020=1027.598,344.293,-136.185,171.737,47.262,159.269
C06021=1027.605,344.540,-136.223,171.743,47.263,159.270
C06022=1027.613,344.788,-136.259,171.750,47.263,159.271
C06023=1027.620,345.035,-136.296,171.756,47.263,159.272
C06024=1027.628,345.282,-136.333,171.762,47.264,159.273
C06025=1027.635,345.529,-136.371,171.769,47.264,159.274
C06026=1027.643,345.776,-136.407,171.775,47.264,159.275
C06027=1027.651,346.023,-136.444,171.781,47.265,159.276
C06028=1027.658,346.270,-136.481,171.788,47.266,159.277
C06029=1027.667,346.518,-136.519,171.794,47.266,159.278
C06030=1027.674,346.765,-136.556,171.801,47.266,159.279
C06031=1027.682,347.012,-136.593,171.807,47.267,159.279
C06032=1027.689,347.259,-136.631,171.813,47.267,159.280
C06033=1027.697,347.506,-136.668,171.820,47.268,159.281
C06034=1027.704,347.753,-136.705,171.826,47.268,159.282
C06035=1027.712,348.000,-136.742,171.833,47.268,159.283
C06036=1027.720,348.247,-136.780,171.839,47.269,159.284
C06037=1027.728,348.494,-136.817,171.845,47.270,159.285
C06038=1027.735,348.741,-136.854,171.852,47.270,159.286
C06039=1027.743,348.989,-136.892,171.859,47.271,159.287
C06040=1027.751,349.235,-136.929,171.866,47.271,159.288
C06041=1027.759,349.483,-136.967,171.872,47.272,159.289
C06042=1027.766,349.730,-137.005,171.878,47.273,159.290
C06043=1027.774,349.977,-137.042,171.885,47.273,159.291
C06044=1027.781,350.193,-137.075,171.891,47.274,159.292
C06045=1027.787,350.409,-137.108,171.896,47.275,159.293
C06046=1027.795,350.626,-137.141,171.902,47.275,159.294
C06047=1027.801,350.842,-137.174,171.908,47.275,159.295
C06048=1027.808,351.058,-137.207,171.914,47.276,159.296
C06049=1027.815,351.275,-137.241,171.920,47.276,159.296
C06050=1027.821,351.491,-137.274,171.925,47.277,159.297
C06051=1027.828,351.707,-137.307,171.931,47.277,159.298
C06052=1027.836,351.954,-137.345,171.938,47.278,159.299
C06053=1027.844,352.201,-137.382,171.944,47.279,159.300
C06054=1027.851,352.448,-137.420,171.951,47.279,159.301
C06055=1027.859,352.695,-137.458,171.958,47.280,159.302
C06056=1027.867,352.942,-137.496,171.965,47.281,159.303
C06057=1027.876,353.190,-137.534,171.971,47.282,159.304
C06058=1027.883,353.436,-137.572,171.978,47.282,159.305
C06059=1027.890,353.683,-137.610,171.985,47.283,159.307
C06060=1027.898,353.930,-137.648,171.992,47.284,159.308
C06061=1027.907,354.177,-137.686,171.999,47.284,159.309
C06062=1027.915,354.424,-137.724,172.005,47.285,159.310
C06063=1027.922,354.671,-137.762,172.012,47.286,159.311
C06064=1027.931,354.918,-137.800,172.019,47.287,159.312
C06065=1027.938,355.165,-137.837,172.026,47.288,159.313
C06066=1027.946,355.412,-137.876,172.032,47.289,159.314
C06067=1027.954,355.659,-137.914,172.040,47.290,159.315
C06068=1027.962,355.906,-137.953,172.047,47.290,159.316
C06069=1027.970,356.152,-137.991,172.053,47.291,159.317
C06070=1027.978,356.400,-138.030,172.060,47.292,159.319
C06071=1027.986,356.647,-138.068,172.067,47.293,159.320
C06072=1027.994,356.893,-138.107,172.074,47.294,159.321
C06073=1028.002,357.141,-138.145,172.081,47.295,159.322
C06074=1028.009,357.387,-138.184,172.088,47.296,159.323
C06075=1028.017,357.634,-138.222,172.095,47.296,159.324
C06076=1028.026,357.882,-138.261,172.102,47.297,159.325
C06077=1028.033,358.128,-138.299,172.108,47.298,159.326
C06078=1028.042,358.375,-138.337,172.116,47.299,159.328
C06079=1028.050,358.622,-138.376,172.123,47.300,159.329
C06080=1028.058,358.868,-138.415,172.130,47.301,159.330
C06081=1028.066,359.115,-138.453,172.137,47.302,159.331
C06082=1028.074,359.362,-138.492,172.144,47.303,159.332
C06083=1028.082,359.609,-138.530,172.151,47.304,159.333
C06084=1028.090,359.856,-138.569,172.158,47.305,159.334
C06085=1028.098,360.103,-138.608,172.165,47.306,159.336
C06086=1028.107,360.350,-138.647,172.172,47.307,159.337
C06087=1028.115,360.597,-138.686,172.179,47.308,159.338
C06088=1028.122,360.843,-138.725,172.187,47.309,159.339
C06089=1028.130,361.090,-138.764,172.194,47.310,159.340
C06090=1028.139,361.337,-138.803,172.201,47.312,159.342
C06091=1028.147,361.584,-138.842,172.208,47.312,159.343
C06092=1028.154,361.831,-138.881,172.216,47.314,159.344
C06093=1028.162,362.077,-138.920,172.222,47.315,159.345
C06094=1028.170,362.324,-138.959,172.230,47.316,159.346
C06095=1028.179,362.571,-138.998,172.237,47.317,159.348
C06096=1028.187,362.818,-139.038,172.244,47.318,159.349
C06097=1028.195,363.065,-139.077,172.252,47.319,159.350
C06098=1028.203,363.311,-139.116,172.258,47.320,159.351
C06099=1028.210,363.558,-139.155,172.266,47.322,159.353
C06100=1028.219,363.805,-139.195,172.274,47.323,159.354
C06101=1028.227,364.052,-139.233,172.281,47.324,159.355
C06102=1028.235,364.298,-139.273,172.288,47.325,159.356
C06103=1028.243,364.545,-139.313,172.295,47.327,159.358
C06104=1028.251,364.765,-139.348,172.302,47.327,159.359
C06105=1028.258,364.984,-139.382,172.309,47.329,159.360
C06106=1028.266,365.204,-139.418,172.315,47.330,159.361
C06107=1028.272,365.424,-139.453,172.322,47.331,159.362
C06108=1028.280,365.643,-139.488,172.328,47.332,159.363
C06109=1028.288,365.862,-139.523,172.335,47.333,159.365
C06110=1028.295,366.082,-139.558,172.342,47.334,159.366
C06111=1028.302,366.302,-139.594,172.348,47.336,159.367
C06112=1028.311,366.549,-139.633,172.356,47.337,159.368
C06113=1028.319,366.795,-139.672,172.363,47.338,159.369
C06114=1028.327,367.042,-139.712,172.371,47.339,159.371
C06115=1028.336,367.289,-139.752,172.379,47.341,159.372
C06116=1028.344,367.535,-139.791,172.386,47.343,159.373
C06117=1028.352,367.782,-139.832,172.394,47.344,159.375
C06118=1028.360,368.028,-139.871,172.402,47.345,159.376
C06119=1028.370,368.276,-139.911,172.409,47.346,159.377
C06120=1028.378,368.522,-139.950,172.416,47.348,159.379
C06121=1028.386,368.768,-139.991,172.424,47.349,159.380
C06122=1028.394,369.015,-140.030,172.431,47.351,159.381
C06123=1028.402,369.262,-140.070,172.439,47.353,159.383
C06124=1028.412,369.509,-140.110,172.447,47.354,159.384
C06125=1028.419,369.755,-140.150,172.454,47.355,159.385
C06126=1028.427,370.002,-140.191,172.462,47.357,159.387
C06127=1028.436,370.248,-140.230,172.470,47.358,159.388
C06128=1028.444,370.495,-140.271,172.477,47.360,159.390
C06129=1028.453,370.741,-140.311,172.485,47.362,159.391
C06130=1028.461,370.988,-140.351,172.493,47.363,159.392
C06131=1028.469,371.235,-140.392,172.501,47.365,159.394
C06132=1028.478,371.481,-140.432,172.509,47.366,159.395
C06133=1028.486,371.728,-140.472,172.516,47.368,159.397
C06134=1028.495,371.974,-140.512,172.524,47.369,159.398
C06135=1028.503,372.221,-140.553,172.533,47.371,159.400
C06136=1028.511,372.467,-140.594,172.541,47.372,159.401
C06137=1028.521,372.714,-140.634,172.549,47.374,159.403
C06138=1028.528,372.961,-140.674,172.557,47.376,159.404
C06139=1028.537,373.207,-140.715,172.564,47.377,159.405
C06140=1028.546,373.454,-140.755,172.572,47.379,159.407
C06141=1028.554,373.700,-140.796,172.580,47.381,159.408
C06142=1028.563,373.947,-140.836,172.588,47.382,159.410
C06143=1028.571,374.193,-140.877,172.596,47.384,159.411
C06144=1028.580,374.440,-140.918,172.604,47.386,159.413
C06145=1028.589,374.686,-140.958,172.612,47.388,159.414
C06146=1028.597,374.933,-140.999,172.620,47.389,159.416
C06147=1028.605,375.179,-141.039,172.628,47.391,159.417
C06148=1028.615,375.425,-141.081,172.636,47.393,159.419
C06149=1028.623,375.672,-141.121,172.645,47.394,159.420
C06150=1028.632,375.919,-141.162,172.653,47.396,159.422
C06151=1028.641,376.165,-141.203,172.661,47.398,159.423
C06152=1028.649,376.412,-141.243,172.669,47.400,159.425
C06153=1028.659,376.658,-141.284,172.677,47.402,159.426
C06154=1028.667,376.905,-141.325,172.686,47.403,159.428
C06155=1028.675,377.151,-141.366,172.693,47.405,159.429
C06156=1028.684,377.397,-141.408,172.701,47.407,159.431
C06157=1028.693,377.644,-141.449,172.709,47.409,159.433
C06158=1028.702,377.890,-141.489,172.719,47.411,159.434
C06159=1028.711,378.137,-141.530,172.727,47.413,159.436
C06160=1028.720,378.383,-141.572,172.735,47.415,159.437
C06161=1028.728,378.629,-141.613,172.743,47.416,159.439
C06162=1028.737,378.876,-141.654,172.752,47.419,159.441
C06163=1028.745,379.122,-141.696,172.760,47.421,159.442
C06164=1028.754,379.352,-141.735,172.768,47.422,159.444
C06165=1028.761,379.582,-141.773,172.776,47.424,159.445
C06166=1028.769,379.812,-141.812,172.783,47.426,159.447
C06167=1028.777,380.042,-141.851,172.791,47.428,159.448
C06168=1028.786,380.273,-141.890,172.799,47.430,159.450
C06169=1028.794,380.503,-141.929,172.807,47.432,159.451
C06170=1028.802,380.733,-141.968,172.815,47.434,159.453
C06171=1028.810,380.963,-142.007,172.823,47.435,159.454
C06172=1028.819,381.209,-142.048,172.831,47.438,159.456
C06173=1028.828,381.456,-142.090,172.839,47.440,159.458
C06174=1028.837,381.702,-142.132,172.849,47.442,159.459
C06175=1028.846,381.948,-142.174,172.857,47.444,159.461
C06176=1028.856,382.194,-142.215,172.866,47.446,159.463
C06177=1028.865,382.441,-142.256,172.874,47.448,159.464
C06178=1028.874,382.687,-142.298,172.883,47.450,159.466
C06179=1028.883,382.934,-142.340,172.892,47.453,159.468
C06180=1028.892,383.180,-142.382,172.901,47.454,159.469
C06181=1028.900,383.426,-142.423,172.909,47.457,159.471
C06182=1028.909,383.673,-142.465,172.918,47.459,159.473
C06183=1028.919,383.918,-142.507,172.926,47.461,159.475
C06184=1028.928,384.165,-142.549,172.936,47.464,159.476
C06185=1028.936,384.411,-142.591,172.944,47.466,159.478
C06186=1028.946,384.657,-142.633,172.953,47.468,159.480
C06187=1028.955,384.903,-142.675,172.962,47.470,159.482
C06188=1028.964,385.150,-142.717,172.971,47.473,159.483
C06189=1028.973,385.396,-142.760,172.980,47.475,159.485
C06190=1028.982,385.642,-142.801,172.988,47.477,159.487
C06191=1028.992,385.888,-142.844,172.998,47.479,159.489
C06192=1029.001,386.134,-142.885,173.006,47.482,159.490
C06193=1029.010,386.380,-142.928,173.015,47.484,159.492
C06194=1029.019,386.627,-142.970,173.024,47.486,159.494
C06195=1029.028,386.873,-143.013,173.033,47.488,159.496
C06196=1029.037,387.119,-143.055,173.042,47.491,159.498
C06197=1029.046,387.365,-143.098,173.052,47.493,159.499
C06198=1029.056,387.612,-143.140,173.060,47.496,159.501
C06199=1029.064,387.858,-143.183,173.069,47.498,159.503
C06200=1029.074,388.104,-143.225,173.079,47.500,159.505
C06201=1029.083,388.350,-143.268,173.087,47.503,159.507
C06202=1029.092,388.596,-143.311,173.097,47.505,159.509
C06203=1029.101,388.842,-143.354,173.106,47.508,159.511
C06204=1029.111,389.088,-143.396,173.115,47.510,159.512
C06205=1029.120,389.334,-143.439,173.124,47.513,159.514
C06206=1029.129,389.581,-143.482,173.133,47.515,159.516
C06207=1029.139,389.827,-143.525,173.143,47.518,159.518
C06208=1029.148,390.073,-143.567,173.153,47.521,159.520
C06209=1029.157,390.318,-143.611,173.161,47.523,159.522
C06210=1029.167,390.565,-143.654,173.170,47.526,159.524
C06211=1029.176,390.811,-143.697,173.180,47.528,159.526
C06212=1029.185,391.057,-143.739,173.190,47.531,159.528
C06213=1029.195,391.303,-143.783,173.199,47.534,159.530
C06214=1029.204,391.549,-143.826,173.209,47.536,159.532
C06215=1029.214,391.794,-143.870,173.217,47.539,159.533
C06216=1029.223,392.041,-143.913,173.227,47.541,159.535
C06217=1029.232,392.287,-143.955,173.236,47.544,159.537
C06218=1029.241,392.533,-143.999,173.246,47.547,159.539
C06219=1029.251,392.780,-144.042,173.256,47.549,159.541
C06220=1029.261,393.025,-144.085,173.265,47.552,159.543
C06221=1029.270,393.271,-144.130,173.275,47.555,159.545
C06222=1029.280,393.517,-144.172,173.285,47.558,159.547
C06223=1029.289,393.763,-144.216,173.294,47.561,159.549
C06224=1029.299,394.012,-144.260,173.304,47.563,159.551
C06225=1029.308,394.262,-144.305,173.314,47.567,159.554
C06226=1029.318,394.513,-144.348,173.324,47.569,159.556
C06227=1029.327,394.763,-144.393,173.334,47.572,159.558
C06228=1029.337,395.009,-144.437,173.343,47.575,159.560
C06229=1029.347,395.255,-144.481,173.353,47.578,159.562
C06230=1029.357,395.501,-144.525,173.363,47.581,159.564
C06231=1029.366,395.747,-144.569,173.372,47.584,159.566
C06232=1029.375,395.992,-144.612,173.382,47.587,159.568
C06233=1029.385,396.238,-144.656,173.392,47.589,159.570
C06234=1029.395,396.484,-144.700,173.403,47.592,159.572
C06235=1029.405,396.730,-144.744,173.412,47.595,159.574
C06236=1029.414,396.976,-144.788,173.422,47.598,159.576
C06237=1029.424,397.222,-144.832,173.432,47.601,159.579
C06238=1029.434,397.468,-144.876,173.442,47.604,159.581
C06239=1029.443,397.714,-144.920,173.452,47.607,159.583
C06240=1029.453,397.959,-144.965,173.462,47.611,159.585
C06241=1029.463,398.205,-145.008,173.473,47.613,159.587
C06242=1029.473,398.451,-145.053,173.483,47.617,159.589
C06243=1029.482,398.697,-145.097,173.492,47.619,159.591
C06244=1029.493,398.943,-145.141,173.502,47.622,159.594
C06245=1029.502,399.188,-145.186,173.513,47.625,159.596
C06246=1029.512,399.434,-145.231,173.523,47.629,159.598
C06247=1029.522,399.679,-145.274,173.533,47.632,159.600
C06248=1029.532,399.926,-145.319,173.543,47.635,159.602
C06249=1029.542,400.172,-145.363,173.554,47.638,159.605
C06250=1029.552,400.417,-145.408,173.564,47.642,159.607
C06251=1029.561,400.663,-145.453,173.574,47.645,159.609
C06252=1029.571,400.908,-145.498,173.585,47.648,159.611
C06253=1029.581,401.153,-145.542,173.595,47.651,159.614
C06254=1029.592,401.400,-145.587,173.606,47.655,159.616
C06255=1029.602,401.645,-145.632,173.616,47.657,159.618
C06256=1029.611,401.891,-145.677,173.627,47.661,159.621
C06257=1029.622,402.137,-145.722,173.638,47.664,159.623
C06258=1029.631,402.382,-145.767,173.648,47.667,159.625
C06259=1029.641,402.628,-145.812,173.658,47.671,159.628
C06260=1029.651,402.874,-145.857,173.669,47.674,159.630
C06261=1029.661,403.120,-145.902,173.679,47.678,159.632
C06262=1029.671,403.365,-145.947,173.691,47.681,159.635
C06263=1029.681,403.611,-145.992,173.701,47.684,159.637
C06264=1029.691,403.856,-146.037,173.712,47.688,159.639
C06265=1029.701,404.102,-146.082,173.722,47.691,159.642
C06266=1029.711,404.347,-146.128,173.733,47.695,159.644
C06267=1029.722,404.594,-146.173,173.744,47.698,159.647
C06268=1029.732,404.838,-146.219,173.755,47.701,159.649
C06269=1029.742,405.085,-146.264,173.766,47.705,159.651
C06270=1029.751,405.330,-146.310,173.776,47.708,159.654
C06271=1029.762,405.576,-146.355,173.788,47.712,159.656
C06272=1029.772,405.822,-146.401,173.798,47.716,159.659
C06273=1029.782,406.067,-146.447,173.809,47.719,159.661
C06274=1029.793,406.313,-146.492,173.820,47.722,159.663
C06275=1029.803,406.558,-146.538,173.831,47.727,159.666
C06276=1029.813,406.803,-146.583,173.842,47.730,159.669
C06277=1029.824,407.050,-146.629,173.854,47.733,159.671
C06278=1029.834,407.295,-146.674,173.865,47.737,159.673
C06279=1029.845,407.541,-146.720,173.875,47.740,159.676
C06280=1029.855,407.786,-146.766,173.887,47.744,159.679
C06281=1029.865,408.031,-146.812,173.898,47.748,159.681
C06282=1029.876,408.277,-146.858,173.910,47.752,159.684
C06283=1029.887,408.522,-146.904,173.921,47.755,159.686
C06284=1029.898,408.794,-146.955,173.933,47.760,159.689
C06285=1029.910,409.066,-147.005,173.946,47.763,159.692
C06286=1029.922,409.337,-147.056,173.959,47.768,159.695
C06287=1029.933,409.609,-147.107,173.971,47.772,159.697
C06288=1029.944,409.854,-147.154,173.982,47.775,159.700
C06289=1029.955,410.100,-147.200,173.994,47.779,159.703
C06290=1029.965,410.345,-147.246,174.005,47.783,159.705
C06291=1029.975,410.591,-147.293,174.017,47.787,159.708
C06292=1029.986,410.836,-147.339,174.029,47.791,159.711
C06293=1029.997,411.081,-147.385,174.040,47.795,159.713
C06294=1030.007,411.327,-147.432,174.052,47.799,159.716
C06295=1030.018,411.572,-147.479,174.064,47.803,159.719
C06296=1030.028,411.819,-147.525,174.075,47.807,159.721
C06297=1030.039,412.064,-147.572,174.087,47.811,159.724
C06298=1030.050,412.309,-147.619,174.099,47.815,159.727
C06299=1030.060,412.554,-147.666,174.110,47.819,159.729
C06300=1030.071,412.799,-147.713,174.122,47.822,159.732
C06301=1030.082,413.045,-147.759,174.135,47.827,159.735
C06302=1030.093,413.290,-147.806,174.147,47.831,159.738
C06303=1030.104,413.535,-147.853,174.158,47.834,159.740
C06304=1030.114,413.781,-147.900,174.170,47.839,159.743
C06305=1030.125,414.026,-147.947,174.182,47.843,159.746
C06306=1030.136,414.272,-147.994,174.195,47.847,159.749
C06307=1030.147,414.517,-148.041,174.207,47.851,159.751
C06308=1030.158,414.762,-148.088,174.219,47.855,159.754
C06309=1030.169,415.008,-148.136,174.231,47.860,159.757
C06310=1030.180,415.253,-148.183,174.243,47.863,159.760
C06311=1030.191,415.499,-148.230,174.255,47.868,159.763
C06312=1030.202,415.743,-148.277,174.267,47.872,159.766
C06313=1030.214,415.989,-148.324,174.280,47.876,159.769
C06314=1030.224,416.234,-148.372,174.292,47.881,159.772
C06315=1030.236,416.479,-148.419,174.305,47.884,159.774
C06316=1030.246,416.724,-148.467,174.317,47.889,159.777
C06317=1030.258,416.969,-148.514,174.329,47.894,159.780
C06318=1030.269,417.215,-148.563,174.342,47.898,159.783
C06319=1030.279,417.460,-148.610,174.354,47.902,159.786
C06320=1030.291,417.705,-148.658,174.367,47.906,159.789
C06321=1030.302,417.950,-148.706,174.379,47.911,159.792
C06322=1030.312,418.195,-148.754,174.393,47.915,159.795
C06323=1030.324,418.440,-148.801,174.405,47.920,159.798
C06324=1030.335,418.685,-148.850,174.418,47.924,159.801
C06325=1030.346,418.931,-148.898,174.431,47.928,159.804
C06326=1030.358,419.176,-148.946,174.443,47.933,159.807
C06327=1030.369,419.421,-148.994,174.457,47.937,159.810
C06328=1030.380,419.666,-149.042,174.470,47.942,159.813
C06329=1030.391,419.911,-149.090,174.482,47.946,159.816
C06330=1030.403,420.156,-149.138,174.495,47.951,159.819
C06331=1030.414,420.401,-149.187,174.509,47.956,159.823
C06332=1030.425,420.646,-149.235,174.521,47.960,159.825
C06333=1030.437,420.891,-149.283,174.534,47.965,159.829
C06334=1030.448,421.137,-149.331,174.547,47.969,159.832
C06335=1030.460,421.382,-149.380,174.561,47.974,159.835
C06336=1030.471,421.627,-149.428,174.574,47.978,159.838
C06337=1030.483,421.871,-149.477,174.588,47.983,159.841
C06338=1030.494,422.117,-149.525,174.601,47.988,159.844
C06339=1030.507,422.362,-149.574,174.613,47.992,159.847
C06340=1030.518,422.607,-149.623,174.627,47.997,159.851
C06341=1030.529,422.852,-149.671,174.640,48.002,159.854
C06342=1030.541,423.097,-149.720,174.654,48.007,159.857
C06343=1030.552,423.341,-149.769,174.667,48.011,159.860
C06344=1030.570,423.704,-149.842,174.688,48.018,159.865
C06345=1030.587,424.065,-149.914,174.708,48.026,159.870
C06346=1030.604,424.428,-149.987,174.729,48.033,159.875
C06347=1030.622,424.788,-150.060,174.749,48.040,159.880
C06348=1030.634,425.034,-150.109,174.762,48.045,159.883
C06349=1030.645,425.279,-150.158,174.776,48.050,159.887
C06350=1030.657,425.524,-150.207,174.790,48.055,159.890
C06351=1030.669,425.768,-150.257,174.804,48.060,159.893
C06352=1030.689,426.178,-150.340,174.827,48.069,159.899
C06353=1030.708,426.588,-150.422,174.851,48.077,159.905
C06354=1030.729,426.998,-150.506,174.875,48.085,159.911
C06355=1030.749,427.407,-150.589,174.898,48.094,159.916
C06356=1030.761,427.652,-150.639,174.913,48.099,159.920
C06357=1030.773,427.896,-150.689,174.927,48.104,159.923
C06358=1030.785,428.141,-150.739,174.942,48.109,159.927
C06359=1030.797,428.385,-150.789,174.956,48.114,159.931
C06360=1030.809,428.631,-150.840,174.971,48.119,159.934
C06361=1030.821,428.875,-150.890,174.985,48.125,159.938
C06362=1030.833,429.120,-150.940,175.000,48.130,159.941
C06363=1030.845,429.364,-150.990,175.015,48.135,159.945
C06364=1030.858,429.609,-151.040,175.029,48.141,159.948
C06365=1030.870,429.854,-151.090,175.044,48.146,159.952
C06366=1030.882,430.098,-151.141,175.059,48.151,159.956
C06367=1030.894,430.343,-151.192,175.074,48.157,159.959
C06368=1030.907,430.588,-151.242,175.089,48.162,159.963
C06369=1030.919,430.832,-151.293,175.104,48.167,159.967
C06370=1030.932,431.077,-151.343,175.119,48.173,159.970
C06371=1030.944,431.321,-151.393,175.133,48.178,159.974
C06372=1030.957,431.566,-151.444,175.148,48.184,159.978
C06373=1030.969,431.810,-151.494,175.164,48.189,159.982
C06374=1030.981,432.055,-151.546,175.179,48.194,159.985
C06375=1030.993,432.299,-151.597,175.194,48.200,159.989
C06376=1031.006,432.543,-151.647,175.209,48.205,159.993
C06377=1031.019,432.788,-151.699,175.225,48.211,159.997
C06378=1031.032,433.032,-151.749,175.240,48.217,160.001
C06379=1031.044,433.277,-151.800,175.256,48.222,160.004
C06380=1031.058,433.522,-151.851,175.271,48.227,160.008
C06381=1031.070,433.766,-151.903,175.287,48.233,160.012
C06382=1031.083,434.011,-151.954,175.303,48.239,160.016
C06383=1031.095,434.255,-152.005,175.318,48.244,160.020
C06384=1031.108,434.499,-152.057,175.334,48.250,160.024
C06385=1031.121,434.744,-152.108,175.350,48.256,160.028
C06386=1031.133,434.988,-152.159,175.366,48.262,160.032
C06387=1031.146,435.233,-152.211,175.382,48.267,160.036
C06388=1031.159,435.477,-152.262,175.397,48.273,160.040
C06389=1031.172,435.721,-152.314,175.414,48.279,160.044
C06390=1031.185,435.966,-152.367,175.430,48.285,160.048
C06391=1031.198,436.210,-152.417,175.445,48.291,160.052
C06392=1031.211,436.455,-152.470,175.462,48.296,160.056
C06393=1031.224,436.699,-152.522,175.478,48.303,160.060
C06394=1031.237,436.942,-152.573,175.494,48.308,160.064
C06395=1031.250,437.187,-152.626,175.510,48.314,160.068
C06396=1031.263,437.431,-152.678,175.527,48.320,160.072
C06397=1031.275,437.675,-152.730,175.544,48.326,160.076
C06398=1031.289,437.920,-152.782,175.560,48.332,160.080
C06399=1031.302,438.163,-152.835,175.577,48.338,160.085
C06400=1031.317,438.427,-152.891,175.595,48.344,160.089
C06401=1031.331,438.690,-152.947,175.613,48.351,160.094
C06402=1031.345,438.953,-153.004,175.631,48.357,160.098
C06403=1031.359,439.216,-153.060,175.649,48.364,160.103
C06404=1031.372,439.460,-153.113,175.666,48.370,160.107
C06405=1031.386,439.704,-153.166,175.683,48.376,160.111
C06406=1031.400,439.949,-153.219,175.700,48.383,160.116
C06407=1031.413,440.193,-153.271,175.717,48.389,160.120
C06408=1031.426,440.437,-153.324,175.734,48.395,160.125
C06409=1031.440,440.680,-153.377,175.751,48.401,160.129
C06410=1031.453,440.924,-153.430,175.768,48.407,160.133
C06411=1031.467,441.168,-153.483,175.786,48.413,160.138
C06412=1031.480,441.412,-153.536,175.803,48.420,160.142
C06413=1031.494,441.657,-153.590,175.822,48.426,160.147
C06414=1031.508,441.900,-153.642,175.839,48.432,160.151
C06415=1031.521,442.144,-153.695,175.856,48.439,160.155
C06416=1031.536,442.388,-153.749,175.874,48.445,160.160
C06417=1031.549,442.632,-153.802,175.892,48.451,160.165
C06418=1031.563,442.876,-153.855,175.909,48.458,160.169
C06419=1031.577,443.120,-153.909,175.927,48.464,160.174
C06420=1031.591,443.363,-153.962,175.945,48.471,160.178
C06421=1031.605,443.606,-154.016,175.963,48.478,160.183
C06422=1031.620,443.849,-154.068,175.981,48.483,160.187
C06423=1031.635,444.093,-154.120,176.000,48.490,160.192
C06424=1031.650,444.336,-154.172,176.018,48.496,160.196
C06425=1031.667,444.579,-154.224,176.035,48.502,160.201
C06426=1031.683,444.823,-154.274,176.054,48.508,160.206
C06427=1031.701,445.067,-154.325,176.073,48.514,160.210
C06428=1031.718,445.311,-154.375,176.091,48.519,160.214
C06429=1031.737,445.555,-154.424,176.109,48.525,160.219
C06430=1031.756,445.798,-154.474,176.129,48.530,160.223
C06431=1031.775,446.042,-154.523,176.147,48.537,160.228
C06432=1031.795,446.287,-154.571,176.167,48.542,160.233
C06433=1031.815,446.531,-154.619,176.185,48.547,160.237
C06434=1031.835,446.775,-154.667,176.205,48.552,160.241
C06435=1031.857,447.020,-154.714,176.224,48.558,160.246
C06436=1031.879,447.264,-154.761,176.243,48.563,160.250
C06437=1031.901,447.509,-154.808,176.262,48.569,160.255
C06438=1031.924,447.753,-154.853,176.281,48.573,160.259
C06439=1031.947,447.998,-154.899,176.301,48.578,160.264
C06440=1031.971,448.243,-154.944,176.320,48.584,160.268
C06441=1031.995,448.487,-154.989,176.340,48.588,160.272
C06442=1032.019,448.733,-155.033,176.360,48.593,160.277
C06443=1032.045,448.977,-155.077,176.379,48.598,160.281
C06444=1032.070,449.223,-155.121,176.399,48.602,160.286
C06445=1032.097,449.468,-155.164,176.419,48.607,160.290
C06446=1032.124,449.713,-155.206,176.440,48.611,160.294
C06447=1032.150,449.958,-155.249,176.460,48.615,160.299
C06448=1032.178,450.204,-155.291,176.480,48.620,160.303
C06449=1032.206,450.449,-155.331,176.501,48.624,160.308
C06450=1032.235,450.694,-155.373,176.520,48.629,160.312
C06451=1032.265,450.939,-155.413,176.541,48.633,160.316
C06452=1032.293,451.185,-155.453,176.562,48.637,160.321
C06453=1032.324,451.431,-155.493,176.583,48.640,160.325
C06454=1032.355,451.675,-155.533,176.603,48.644,160.329
C06455=1032.386,451.921,-155.571,176.624,48.648,160.334
C06456=1032.418,452.167,-155.609,176.645,48.652,160.338
C06457=1032.450,452.413,-155.648,176.666,48.656,160.342
C06458=1032.483,452.658,-155.685,176.687,48.660,160.347
C06459=1032.516,452.903,-155.722,176.708,48.664,160.351
C06460=1032.573,453.314,-155.783,176.745,48.669,160.358
C06461=1032.290,453.381,-156.114,176.748,48.734,160.379
C06462=1032.239,453.015,-156.060,176.715,48.730,160.373
C06463=1032.206,452.770,-156.023,176.695,48.726,160.368
C06464=1032.173,452.524,-155.986,176.673,48.722,160.364
C06465=1032.141,452.279,-155.948,176.652,48.718,160.360
C06466=1032.109,452.033,-155.910,176.631,48.715,160.355
C06467=1032.077,451.787,-155.872,176.610,48.711,160.351
C06468=1032.046,451.542,-155.832,176.589,48.708,160.347
C06469=1032.016,451.297,-155.793,176.568,48.704,160.342
C06470=1031.986,451.051,-155.752,176.548,48.700,160.338
C06471=1031.956,450.806,-155.712,176.527,48.696,160.334
C06472=1031.927,450.560,-155.672,176.506,48.692,160.329
C06473=1031.899,450.315,-155.631,176.486,48.687,160.325
C06474=1031.871,450.070,-155.589,176.465,48.683,160.321
C06475=1031.844,449.824,-155.547,176.445,48.679,160.316
C06476=1031.817,449.579,-155.504,176.425,48.674,160.312
C06477=1031.790,449.334,-155.462,176.406,48.670,160.307
C06478=1031.764,449.088,-155.419,176.385,48.666,160.303
C06479=1031.738,448.845,-155.375,176.366,48.661,160.299
C06480=1031.713,448.599,-155.331,176.346,48.656,160.294
C06481=1031.689,448.354,-155.286,176.326,48.652,160.290
C06482=1031.665,448.110,-155.241,176.306,48.647,160.285
C06483=1031.641,447.865,-155.196,176.287,48.642,160.281
C06484=1031.619,447.620,-155.150,176.267,48.637,160.277
C06485=1031.597,447.375,-155.104,176.247,48.632,160.272
C06486=1031.574,447.131,-155.058,176.229,48.627,160.268
C06487=1031.553,446.886,-155.010,176.209,48.622,160.263
C06488=1031.531,446.642,-154.963,176.190,48.616,160.259
C06489=1031.511,446.398,-154.916,176.171,48.612,160.254
C06490=1031.491,446.153,-154.867,176.152,48.606,160.250
C06491=1031.471,445.909,-154.819,176.133,48.601,160.245
C06492=1031.452,445.665,-154.770,176.114,48.595,160.241
C06493=1031.434,445.421,-154.720,176.095,48.590,160.236
C06494=1031.416,445.178,-154.671,176.077,48.584,160.232
C06495=1031.398,444.934,-154.620,176.059,48.578,160.228
C06496=1031.381,444.689,-154.569,176.039,48.572,160.223
C06497=1031.364,444.446,-154.518,176.021,48.566,160.218
C06498=1031.348,444.203,-154.467,176.003,48.560,160.214
C06499=1031.333,443.959,-154.415,175.985,48.554,160.209
C06500=1031.318,443.715,-154.362,175.967,48.548,160.205
C06501=1031.303,443.472,-154.310,175.948,48.542,160.200
C06502=1031.289,443.230,-154.257,175.931,48.535,160.196
C06503=1031.275,442.986,-154.203,175.913,48.530,160.191
C06504=1031.262,442.742,-154.150,175.895,48.523,160.186
C06505=1031.247,442.499,-154.096,175.877,48.517,160.182
C06506=1031.234,442.255,-154.043,175.859,48.511,160.178
C06507=1031.219,442.010,-153.990,175.842,48.504,160.173
C06508=1031.206,441.766,-153.937,175.823,48.498,160.169
C06509=1031.193,441.523,-153.883,175.806,48.492,160.164
C06510=1031.179,441.279,-153.830,175.789,48.486,160.160
C06511=1031.165,441.035,-153.777,175.772,48.479,160.155
C06512=1031.151,440.791,-153.724,175.754,48.473,160.151
C06513=1031.138,440.547,-153.671,175.737,48.467,160.146
C06514=1031.125,440.303,-153.619,175.719,48.461,160.142
C06515=1031.112,440.059,-153.566,175.702,48.455,160.138
C06516=1031.098,439.815,-153.513,175.685,48.449,160.133
C06517=1031.085,439.571,-153.460,175.668,48.443,160.129
C06518=1031.071,439.327,-153.408,175.652,48.436,160.125
C06519=1031.057,439.063,-153.350,175.633,48.430,160.120
C06520=1031.042,438.799,-153.294,175.615,48.424,160.116
C06521=1031.029,438.535,-153.238,175.596,48.417,160.111
C06522=1031.013,438.271,-153.180,175.579,48.411,160.107
C06523=1031.000,438.026,-153.128,175.562,48.405,160.102
C06524=1030.988,437.783,-153.076,175.545,48.399,160.098
C06525=1030.975,437.538,-153.024,175.528,48.394,160.094
C06526=1030.961,437.294,-152.972,175.512,48.387,160.090
C06527=1030.948,437.049,-152.920,175.496,48.382,160.086
C06528=1030.935,436.806,-152.868,175.480,48.375,160.082
C06529=1030.922,436.561,-152.816,175.463,48.370,160.078
C06530=1030.909,436.317,-152.764,175.447,48.364,160.074
C06531=1030.896,436.073,-152.712,175.430,48.358,160.069
C06532=1030.883,435.829,-152.660,175.415,48.352,160.065
C06533=1030.870,435.584,-152.608,175.398,48.347,160.062
C06534=1030.857,435.340,-152.557,175.382,48.341,160.057
C06535=1030.844,435.095,-152.506,175.366,48.336,160.053
C06536=1030.832,434.851,-152.454,175.350,48.330,160.050
C06537=1030.819,434.606,-152.402,175.335,48.324,160.046
C06538=1030.806,434.363,-152.351,175.318,48.319,160.042
C06539=1030.793,434.118,-152.299,175.303,48.313,160.038
C06540=1030.781,433.873,-152.248,175.287,48.308,160.034
C06541=1030.768,433.630,-152.197,175.272,48.302,160.030
C06542=1030.755,433.385,-152.145,175.256,48.296,160.026
C06543=1030.743,433.140,-152.094,175.240,48.291,160.022
C06544=1030.730,432.896,-152.043,175.225,48.286,160.018
C06545=1030.717,432.651,-151.992,175.209,48.280,160.015
C06546=1030.704,432.406,-151.942,175.194,48.275,160.011
C06547=1030.692,432.162,-151.891,175.179,48.269,160.007
C06548=1030.679,431.918,-151.841,175.163,48.264,160.003
C06549=1030.666,431.673,-151.789,175.148,48.259,160.000
C06550=1030.654,431.428,-151.739,175.133,48.253,159.996
C06551=1030.642,431.184,-151.688,175.118,48.248,159.992
C06552=1030.629,430.940,-151.637,175.103,48.243,159.988
C06553=1030.617,430.695,-151.587,175.088,48.237,159.985
C06554=1030.605,430.450,-151.537,175.073,48.232,159.981
C06555=1030.592,430.206,-151.486,175.058,48.227,159.977
C06556=1030.580,429.961,-151.436,175.043,48.221,159.974
C06557=1030.567,429.717,-151.385,175.028,48.216,159.970
C06558=1030.555,429.472,-151.334,175.014,48.211,159.966
C06559=1030.544,429.227,-151.285,174.999,48.206,159.963
C06560=1030.531,428.983,-151.235,174.984,48.201,159.959
C06561=1030.519,428.738,-151.185,174.970,48.195,159.956
C06562=1030.507,428.493,-151.134,174.955,48.190,159.952
C06563=1030.494,428.248,-151.084,174.941,48.185,159.949
C06564=1030.483,428.004,-151.035,174.926,48.180,159.945
C06565=1030.471,427.759,-150.984,174.912,48.175,159.942
C06566=1030.459,427.514,-150.934,174.897,48.170,159.938
C06567=1030.447,427.270,-150.884,174.883,48.165,159.935
C06568=1030.435,427.025,-150.834,174.869,48.160,159.931
C06569=1030.423,426.780,-150.785,174.855,48.155,159.928
C06570=1030.411,426.536,-150.735,174.840,48.150,159.924
C06571=1030.399,426.290,-150.686,174.826,48.145,159.921
C06572=1030.387,426.046,-150.636,174.813,48.140,159.917
C06573=1030.375,425.801,-150.586,174.798,48.135,159.914
C06574=1030.364,425.556,-150.537,174.784,48.130,159.911
C06575=1030.351,425.311,-150.488,174.770,48.125,159.907
C06576=1030.340,425.067,-150.439,174.755,48.120,159.904
C06577=1030.328,424.821,-150.390,174.742,48.116,159.901
C06578=1030.316,424.577,-150.340,174.728,48.111,159.897
C06579=1030.303,424.293,-150.283,174.712,48.105,159.893
C06580=1030.288,424.008,-150.226,174.697,48.100,159.890
C06581=1030.275,423.724,-150.169,174.680,48.094,159.886
C06582=1030.262,423.440,-150.112,174.665,48.088,159.882
C06583=1030.250,423.196,-150.063,174.652,48.084,159.879
C06584=1030.238,422.950,-150.014,174.638,48.079,159.875
C06585=1030.227,422.705,-149.965,174.624,48.075,159.872
C06586=1030.216,422.460,-149.917,174.610,48.070,159.869
C06587=1030.204,422.215,-149.868,174.597,48.065,159.866
C06588=1030.192,421.970,-149.820,174.584,48.060,159.863
C06589=1030.180,421.725,-149.771,174.571,48.056,159.859
C06590=1030.169,421.479,-149.722,174.558,48.052,159.856
C06591=1030.157,421.235,-149.674,174.544,48.047,159.853
C06592=1030.146,420.990,-149.626,174.531,48.043,159.850
C06593=1030.135,420.745,-149.577,174.518,48.038,159.847
C06594=1030.123,420.500,-149.529,174.504,48.033,159.844
C06595=1030.112,420.254,-149.481,174.491,48.029,159.841
C06596=1030.100,420.010,-149.432,174.479,48.025,159.838
C06597=1030.088,419.765,-149.384,174.466,48.020,159.835
C06598=1030.077,419.519,-149.336,174.452,48.016,159.831
C06599=1030.060,419.140,-149.262,174.433,48.009,159.827
C06600=1030.043,418.761,-149.187,174.412,48.003,159.822
C06601=1030.025,418.381,-149.113,174.393,47.995,159.817
C06602=1030.008,418.001,-149.039,174.374,47.989,159.813
C06603=1029.997,417.757,-148.991,174.360,47.984,159.810
C06604=1029.986,417.511,-148.943,174.347,47.980,159.807
C06605=1029.975,417.266,-148.895,174.335,47.976,159.804
C06606=1029.964,417.021,-148.847,174.322,47.972,159.801
C06607=1029.953,416.775,-148.800,174.310,47.967,159.798
C06608=1029.942,416.531,-148.752,174.297,47.963,159.795
C06609=1029.931,416.285,-148.705,174.285,47.959,159.792
C06610=1029.920,416.040,-148.657,174.273,47.955,159.790
C06611=1029.909,415.795,-148.610,174.260,47.951,159.787
C06612=1029.897,415.549,-148.563,174.248,47.946,159.784
C06613=1029.887,415.304,-148.515,174.235,47.942,159.781
C06614=1029.875,415.059,-148.468,174.224,47.938,159.778
C06615=1029.865,414.814,-148.421,174.212,47.934,159.775
C06616=1029.853,414.568,-148.374,174.199,47.930,159.772
C06617=1029.842,414.323,-148.327,174.187,47.926,159.769
C06618=1029.832,414.077,-148.280,174.175,47.922,159.767
C06619=1029.821,413.832,-148.233,174.162,47.918,159.764
C06620=1029.811,413.587,-148.186,174.150,47.914,159.761
C06621=1029.799,413.341,-148.139,174.139,47.910,159.758
C06622=1029.788,413.096,-148.092,174.127,47.906,159.756
C06623=1029.778,412.851,-148.045,174.115,47.902,159.753
C06624=1029.767,412.606,-147.998,174.102,47.898,159.750
C06625=1029.755,412.360,-147.951,174.091,47.894,159.747
C06626=1029.745,412.115,-147.904,174.079,47.891,159.745
C06627=1029.735,411.869,-147.858,174.067,47.887,159.742
C06628=1029.724,411.624,-147.811,174.056,47.883,159.739
C06629=1029.714,411.379,-147.764,174.044,47.879,159.737
C06630=1029.703,411.133,-147.718,174.032,47.875,159.734
C06631=1029.693,410.888,-147.671,174.021,47.871,159.731
C06632=1029.682,410.642,-147.625,174.009,47.867,159.729
C06633=1029.671,410.396,-147.578,173.998,47.864,159.726
C06634=1029.661,410.151,-147.532,173.986,47.860,159.723
C06635=1029.644,409.767,-147.459,173.967,47.854,159.719
C06636=1029.627,409.382,-147.388,173.950,47.848,159.715
C06637=1029.610,408.997,-147.315,173.931,47.843,159.711
C06638=1029.594,408.612,-147.244,173.914,47.837,159.707
C06639=1029.583,408.366,-147.198,173.902,47.833,159.705
C06640=1029.573,408.121,-147.152,173.891,47.830,159.702
C06641=1029.563,407.875,-147.105,173.880,47.826,159.700
C06642=1029.552,407.629,-147.059,173.868,47.823,159.697
C06643=1029.542,407.384,-147.014,173.858,47.819,159.695
C06644=1029.532,407.139,-146.968,173.846,47.815,159.692
C06645=1029.521,406.893,-146.922,173.835,47.812,159.690
C06646=1029.510,406.648,-146.876,173.824,47.808,159.687
C06647=1029.501,406.402,-146.831,173.813,47.805,159.685
C06648=1029.490,406.156,-146.785,173.802,47.801,159.682
C06649=1029.479,405.911,-146.740,173.791,47.798,159.680
C06650=1029.470,405.665,-146.695,173.779,47.795,159.677
C06651=1029.459,405.420,-146.649,173.769,47.791,159.675
C06652=1029.449,405.174,-146.604,173.758,47.788,159.672
C06653=1029.439,404.929,-146.558,173.747,47.784,159.670
C06654=1029.428,404.682,-146.513,173.736,47.781,159.668
C06655=1029.418,404.438,-146.467,173.725,47.778,159.665
C06656=1029.408,404.191,-146.422,173.715,47.774,159.663
C06657=1029.398,403.946,-146.377,173.704,47.770,159.660
C06658=1029.388,403.700,-146.331,173.694,47.767,159.658
C06659=1029.378,403.455,-146.287,173.682,47.764,159.656
C06660=1029.368,403.210,-146.241,173.671,47.761,159.654
C06661=1029.358,402.964,-146.196,173.661,47.757,159.651
C06662=1029.348,402.718,-146.151,173.650,47.754,159.649
C06663=1029.338,402.473,-146.106,173.640,47.751,159.646
C06664=1029.329,402.226,-146.060,173.630,47.748,159.644
C06665=1029.319,401.981,-146.016,173.618,47.744,159.642
C06666=1029.308,401.735,-145.971,173.608,47.741,159.640
C06667=1029.298,401.489,-145.926,173.597,47.738,159.637
C06668=1029.288,401.244,-145.881,173.587,47.734,159.635
C06669=1029.279,400.998,-145.837,173.576,47.732,159.633
C06670=1029.269,400.753,-145.792,173.566,47.728,159.630
C06671=1029.259,400.506,-145.747,173.556,47.725,159.628
C06672=1029.249,400.261,-145.703,173.545,47.722,159.626
C06673=1029.239,400.015,-145.658,173.535,47.719,159.624
C06674=1029.229,399.769,-145.613,173.525,47.716,159.622
C06675=1029.220,399.523,-145.569,173.514,47.713,159.619
C06676=1029.210,399.278,-145.524,173.504,47.710,159.617
C06677=1029.199,399.033,-145.480,173.494,47.707,159.615
C06678=1029.190,398.787,-145.436,173.483,47.704,159.613
C06679=1029.180,398.540,-145.391,173.473,47.701,159.610
C06680=1029.170,398.294,-145.347,173.464,47.698,159.608
C06681=1029.160,398.048,-145.303,173.454,47.695,159.606
C06682=1029.150,397.803,-145.259,173.443,47.692,159.604
C06683=1029.140,397.557,-145.215,173.433,47.689,159.602
C06684=1029.131,397.311,-145.171,173.423,47.686,159.600
C06685=1029.120,397.066,-145.127,173.413,47.683,159.598
C06686=1029.111,396.820,-145.083,173.403,47.681,159.596
C06687=1029.102,396.573,-145.038,173.393,47.677,159.593
C06688=1029.092,396.328,-144.995,173.383,47.675,159.591
C06689=1029.083,396.082,-144.951,173.373,47.672,159.589
C06690=1029.073,395.836,-144.907,173.363,47.669,159.587
C06691=1029.063,395.590,-144.864,173.353,47.666,159.585
C06692=1029.054,395.344,-144.819,173.344,47.663,159.583
C06693=1029.044,395.098,-144.776,173.334,47.660,159.581
C06694=1029.035,394.853,-144.732,173.324,47.657,159.579
C06695=1029.025,394.601,-144.687,173.314,47.655,159.577
C06696=1029.015,394.348,-144.642,173.304,47.652,159.575
C06697=1029.005,394.096,-144.598,173.294,47.649,159.573
C06698=1028.995,393.843,-144.553,173.284,47.646,159.571
C06699=1028.986,393.598,-144.509,173.275,47.644,159.569
C06700=1028.976,393.351,-144.466,173.265,47.641,159.567
C06701=1028.967,393.105,-144.422,173.256,47.638,159.565
C06702=1028.958,392.860,-144.380,173.246,47.636,159.563
C06703=1028.948,392.613,-144.336,173.236,47.633,159.561
C06704=1028.938,392.368,-144.292,173.227,47.631,159.559
C06705=1028.929,392.122,-144.250,173.217,47.628,159.557
C06706=1028.920,391.875,-144.206,173.207,47.625,159.555
C06707=1028.910,391.629,-144.163,173.198,47.623,159.553
C06708=1028.901,391.383,-144.120,173.188,47.620,159.551
C06709=1028.891,391.137,-144.076,173.179,47.617,159.549
C06710=1028.882,390.892,-144.034,173.169,47.615,159.547
C06711=1028.873,390.645,-143.991,173.160,47.613,159.545
C06712=1028.863,390.400,-143.947,173.151,47.610,159.543
C06713=1028.854,390.153,-143.904,173.142,47.607,159.541
C06714=1028.845,389.907,-143.862,173.132,47.605,159.539
C06715=1028.836,389.662,-143.819,173.122,47.602,159.537
C06716=1028.827,389.415,-143.776,173.113,47.600,159.535
C06717=1028.817,389.169,-143.733,173.104,47.597,159.533
C06718=1028.807,388.923,-143.691,173.095,47.595,159.532
C06719=1028.799,388.677,-143.648,173.086,47.593,159.530
C06720=1028.790,388.431,-143.605,173.076,47.590,159.528
C06721=1028.780,388.184,-143.562,173.067,47.588,159.526
C06722=1028.771,387.939,-143.520,173.058,47.585,159.524
C06723=1028.762,387.693,-143.477,173.049,47.583,159.522
C06724=1028.752,387.446,-143.434,173.040,47.581,159.521
C06725=1028.743,387.200,-143.392,173.031,47.579,159.519
C06726=1028.734,386.954,-143.350,173.022,47.576,159.517
C06727=1028.726,386.708,-143.307,173.013,47.574,159.515
C06728=1028.716,386.461,-143.265,173.003,47.572,159.513
C06729=1028.707,386.215,-143.222,172.995,47.569,159.512
C06730=1028.698,385.969,-143.180,172.986,47.567,159.510
C06731=1028.688,385.722,-143.138,172.977,47.565,159.508
C06732=1028.679,385.476,-143.096,172.968,47.563,159.506
C06733=1028.670,385.230,-143.054,172.959,47.561,159.504
C06734=1028.661,384.984,-143.012,172.950,47.558,159.503
C06735=1028.652,384.738,-142.970,172.941,47.556,159.501
C06736=1028.643,384.492,-142.928,172.932,47.554,159.499
C06737=1028.634,384.245,-142.886,172.924,47.551,159.497
C06738=1028.624,383.999,-142.843,172.915,47.550,159.496
C06739=1028.615,383.753,-142.802,172.906,47.548,159.494
C06740=1028.606,383.506,-142.760,172.897,47.545,159.492
C06741=1028.597,383.260,-142.718,172.888,47.543,159.491
C06742=1028.588,383.014,-142.676,172.880,47.541,159.489
C06743=1028.579,382.768,-142.634,172.871,47.539,159.487
C06744=1028.570,382.521,-142.592,172.862,47.537,159.486
C06745=1028.560,382.275,-142.551,172.853,47.535,159.484
C06746=1028.551,382.029,-142.509,172.845,47.533,159.482
C06747=1028.543,381.783,-142.468,172.836,47.531,159.480
C06748=1028.534,381.536,-142.426,172.828,47.529,159.479
C06749=1028.525,381.291,-142.385,172.819,47.527,159.477
C06750=1028.516,381.044,-142.343,172.811,47.525,159.476
C06751=1028.508,380.813,-142.304,172.803,47.523,159.474
C06752=1028.500,380.581,-142.264,172.795,47.521,159.473
C06753=1028.492,380.350,-142.225,172.787,47.519,159.471
C06754=1028.483,380.118,-142.187,172.779,47.518,159.469
C06755=1028.475,379.888,-142.148,172.771,47.516,159.468
C06756=1028.467,379.657,-142.109,172.763,47.514,159.466
C06757=1028.459,379.425,-142.070,172.755,47.512,159.465
C06758=1028.451,379.195,-142.031,172.747,47.510,159.463
C06759=1028.442,378.948,-141.990,172.738,47.509,159.462
C06760=1028.433,378.702,-141.948,172.730,47.507,159.460
C06761=1028.425,378.455,-141.907,172.722,47.504,159.458
C06762=1028.416,378.209,-141.866,172.713,47.503,159.457
C06763=1028.407,377.963,-141.824,172.705,47.501,159.455
C06764=1028.399,377.716,-141.783,172.697,47.499,159.454
C06765=1028.390,377.470,-141.742,172.688,47.498,159.452
C06766=1028.382,377.223,-141.701,172.680,47.496,159.451
C06767=1028.372,376.977,-141.660,172.672,47.494,159.449
C06768=1028.364,376.731,-141.619,172.664,47.492,159.448
C06769=1028.355,376.484,-141.578,172.655,47.490,159.446
C06770=1028.346,376.237,-141.538,172.647,47.489,159.445
C06771=1028.338,375.991,-141.496,172.639,47.487,159.443
C06772=1028.328,375.745,-141.456,172.630,47.485,159.441
C06773=1028.320,375.498,-141.415,172.622,47.483,159.440
C06774=1028.312,375.251,-141.374,172.615,47.482,159.439
C06775=1028.302,375.005,-141.334,172.607,47.480,159.437
C06776=1028.294,374.758,-141.293,172.598,47.479,159.436
C06777=1028.286,374.511,-141.252,172.590,47.477,159.434
C06778=1028.277,374.265,-141.212,172.582,47.475,159.433
C06779=1028.268,374.018,-141.171,172.574,47.474,159.431
C06780=1028.259,373.772,-141.131,172.566,47.472,159.430
C06781=1028.251,373.525,-141.090,172.559,47.470,159.428
C06782=1028.243,373.279,-141.049,172.550,47.469,159.427
C06783=1028.234,373.033,-141.009,172.542,47.467,159.425
C06784=1028.225,372.786,-140.968,172.534,47.466,159.424
C06785=1028.217,372.540,-140.928,172.526,47.464,159.422
C06786=1028.208,372.293,-140.887,172.519,47.463,159.421
C06787=1028.200,372.046,-140.847,172.511,47.461,159.419
C06788=1028.192,371.800,-140.807,172.503,47.459,159.418
C06789=1028.183,371.553,-140.766,172.494,47.458,159.417
C06790=1028.175,371.307,-140.726,172.487,47.457,159.415
C06791=1028.166,371.060,-140.686,172.479,47.455,159.414
C06792=1028.158,370.813,-140.645,172.471,47.453,159.412
C06793=1028.149,370.567,-140.606,172.463,47.452,159.411
C06794=1028.141,370.321,-140.565,172.456,47.451,159.410
C06795=1028.133,370.074,-140.525,172.448,47.449,159.408
C06796=1028.124,369.827,-140.485,172.440,47.448,159.407
C06797=1028.116,369.581,-140.445,172.433,47.446,159.406
C06798=1028.108,369.334,-140.405,172.425,47.445,159.404
C06799=1028.100,369.088,-140.365,172.417,47.443,159.403
C06800=1028.092,368.841,-140.325,172.409,47.442,159.401
C06801=1028.083,368.594,-140.285,172.402,47.441,159.400
C06802=1028.074,368.348,-140.245,172.394,47.439,159.399
C06803=1028.066,368.101,-140.206,172.387,47.438,159.397
C06804=1028.058,367.854,-140.166,172.379,47.437,159.396
C06805=1028.050,367.608,-140.126,172.371,47.435,159.395
C06806=1028.041,367.361,-140.087,172.364,47.434,159.393
C06807=1028.033,367.113,-140.047,172.356,47.433,159.392
C06808=1028.024,366.867,-140.007,172.348,47.431,159.391
C06809=1028.016,366.621,-139.967,172.341,47.430,159.389
C06810=1028.007,366.374,-139.928,172.333,47.429,159.388
C06811=1028.001,366.154,-139.892,172.327,47.428,159.387
C06812=1027.993,365.933,-139.857,172.320,47.427,159.386
C06813=1027.985,365.712,-139.822,172.313,47.426,159.385
C06814=1027.978,365.491,-139.787,172.307,47.425,159.383
C06815=1027.970,365.271,-139.752,172.300,47.424,159.382
C06816=1027.964,365.050,-139.716,172.293,47.423,159.381
C06817=1027.956,364.829,-139.681,172.286,47.421,159.380
C06818=1027.949,364.609,-139.646,172.280,47.420,159.379
C06819=1027.940,364.362,-139.607,172.273,47.420,159.378
C06820=1027.932,364.116,-139.567,172.265,47.418,159.376
C06821=1027.924,363.869,-139.527,172.258,47.417,159.375
C06822=1027.916,363.621,-139.489,172.250,47.416,159.374
C06823=1027.907,363.375,-139.449,172.244,47.415,159.373
C06824=1027.900,363.128,-139.410,172.236,47.413,159.371
C06825=1027.891,362.881,-139.370,172.229,47.413,159.370
C06826=1027.884,362.635,-139.332,172.221,47.411,159.369
C06827=1027.875,362.388,-139.293,172.214,47.411,159.368
C06828=1027.867,362.141,-139.253,172.206,47.409,159.366
C06829=1027.859,361.894,-139.214,172.200,47.408,159.365
C06830=1027.851,361.648,-139.175,172.192,47.407,159.364
C06831=1027.843,361.400,-139.136,172.185,47.406,159.363
C06832=1027.836,361.154,-139.097,172.177,47.405,159.362
C06833=1027.827,360.907,-139.058,172.171,47.404,159.361
C06834=1027.819,360.660,-139.019,172.164,47.403,159.359
C06835=1027.811,360.413,-138.980,172.156,47.402,159.358
C06836=1027.803,360.167,-138.942,172.149,47.401,159.357
C06837=1027.795,359.920,-138.903,172.143,47.400,159.356
C06838=1027.787,359.673,-138.864,172.135,47.400,159.355
C06839=1027.779,359.426,-138.825,172.128,47.398,159.353
C06840=1027.771,359.180,-138.786,172.120,47.397,159.352
C06841=1027.763,358.932,-138.748,172.114,47.396,159.351
C06842=1027.754,358.685,-138.709,172.107,47.396,159.350
C06843=1027.747,358.439,-138.671,172.099,47.395,159.349
C06844=1027.739,358.192,-138.632,172.092,47.394,159.348
C06845=1027.731,357.944,-138.594,172.086,47.393,159.347
C06846=1027.723,357.698,-138.555,172.078,47.392,159.345
C06847=1027.715,357.451,-138.517,172.071,47.391,159.344
C06848=1027.707,357.203,-138.478,172.065,47.390,159.343
C06849=1027.699,356.957,-138.440,172.057,47.389,159.342
C06850=1027.691,356.710,-138.401,172.050,47.389,159.341
C06851=1027.683,356.463,-138.363,172.044,47.388,159.340
C06852=1027.675,356.216,-138.325,172.037,47.388,159.339
C06853=1027.667,355.970,-138.287,172.029,47.387,159.338
C06854=1027.659,355.722,-138.248,172.023,47.386,159.337
C06855=1027.651,355.475,-138.210,172.016,47.385,159.336
C06856=1027.643,355.229,-138.171,172.009,47.384,159.334
C06857=1027.635,354.982,-138.133,172.002,47.383,159.333
C06858=1027.628,354.734,-138.095,171.995,47.383,159.332
C06859=1027.620,354.487,-138.057,171.989,47.382,159.331
C06860=1027.611,354.241,-138.019,171.982,47.382,159.330
C06861=1027.604,353.994,-137.981,171.974,47.381,159.329
C06862=1027.596,353.747,-137.943,171.968,47.380,159.328
C06863=1027.588,353.500,-137.905,171.961,47.380,159.327
C06864=1027.580,353.253,-137.867,171.955,47.379,159.326
C06865=1027.572,353.006,-137.829,171.948,47.378,159.325
C06866=1027.564,352.758,-137.791,171.941,47.378,159.324
C06867=1027.556,352.512,-137.754,171.934,47.377,159.323
C06868=1027.549,352.265,-137.716,171.927,47.377,159.322
C06869=1027.541,352.018,-137.677,171.921,47.376,159.321
C06870=1027.533,351.771,-137.640,171.914,47.375,159.320
C06871=1027.526,351.554,-137.607,171.908,47.375,159.319
C06872=1027.519,351.336,-137.574,171.902,47.374,159.318
C06873=1027.513,351.119,-137.540,171.897,47.373,159.317
C06874=1027.506,350.901,-137.507,171.891,47.373,159.316
C06875=1027.499,350.684,-137.474,171.885,47.372,159.315
C06876=1027.492,350.466,-137.440,171.879,47.372,159.314
C06877=1027.485,350.249,-137.408,171.873,47.372,159.314
C06878=1027.478,350.032,-137.374,171.867,47.371,159.313
C06879=1027.471,349.785,-137.337,171.861,47.371,159.312
C06880=1027.464,349.538,-137.299,171.854,47.370,159.311
C06881=1027.455,349.291,-137.261,171.848,47.370,159.310
C06882=1027.447,349.044,-137.224,171.841,47.370,159.309
C06883=1027.440,348.796,-137.186,171.834,47.368,159.308
C06884=1027.432,348.550,-137.149,171.827,47.368,159.307
C06885=1027.425,348.303,-137.112,171.821,47.368,159.306
C06886=1027.417,348.055,-137.074,171.815,47.367,159.305
C06887=1027.409,347.808,-137.037,171.808,47.367,159.304
C06888=1027.402,347.561,-136.999,171.802,47.366,159.303
C06889=1027.394,347.314,-136.963,171.795,47.366,159.302
C06890=1027.386,347.067,-136.926,171.789,47.366,159.301
C06891=1027.379,346.820,-136.888,171.782,47.366,159.300
C06892=1027.370,346.572,-136.851,171.776,47.365,159.299
C06893=1027.363,346.325,-136.813,171.769,47.365,159.298
C06894=1027.355,346.078,-136.776,171.763,47.365,159.297
C06895=1027.348,345.831,-136.739,171.757,47.364,159.297
C06896=1027.340,345.584,-136.703,171.750,47.364,159.296
C06897=1027.333,345.337,-136.665,171.744,47.364,159.295
C06898=1027.325,345.090,-136.628,171.737,47.363,159.294
C06899=1027.318,344.843,-136.591,171.731,47.363,159.293
C06900=1027.310,344.595,-136.554,171.725,47.363,159.292
C06901=1027.302,344.348,-136.517,171.718,47.362,159.291
C06902=1027.295,344.101,-136.480,171.712,47.362,159.290
C06903=1027.287,343.854,-136.444,171.705,47.362,159.289
C06904=1027.280,343.607,-136.406,171.699,47.361,159.288
C06905=1027.272,343.360,-136.369,171.693,47.361,159.288
C06906=1027.264,343.113,-136.333,171.686,47.361,159.287
C06907=1027.257,342.865,-136.295,171.681,47.361,159.286
C06908=1027.249,342.618,-136.259,171.675,47.361,159.285
C06909=1027.242,342.371,-136.222,171.668,47.361,159.284
C06910=1027.234,342.123,-136.186,171.662,47.360,159.283
C06911=1027.226,341.877,-136.149,171.656,47.360,159.282
C06912=1027.219,341.629,-136.112,171.649,47.360,159.282
C06913=1027.212,341.383,-136.075,171.643,47.360,159.281
C06914=1027.204,341.135,-136.039,171.637,47.359,159.280
C06915=1027.197,340.887,-136.002,171.631,47.360,159.279
C06916=1027.189,340.641,-135.965,171.625,47.359,159.278
C06917=1027.182,340.393,-135.929,171.619,47.359,159.277
C06918=1027.175,340.145,-135.892,171.613,47.359,159.277
C06919=1027.167,339.899,-135.856,171.606,47.359,159.276
C06920=1027.160,339.652,-135.819,171.600,47.359,159.275
C06921=1027.152,339.404,-135.783,171.594,47.359,159.274
C06922=1027.144,339.157,-135.747,171.587,47.358,159.273
C06923=1027.137,338.910,-135.711,171.582,47.359,159.272
C06924=1027.129,338.663,-135.674,171.576,47.359,159.272
C06925=1027.122,338.416,-135.638,171.569,47.359,159.271
C06926=1027.114,338.168,-135.602,171.563,47.359,159.270
C06927=1027.107,337.921,-135.565,171.557,47.358,159.269
C06928=1027.099,337.673,-135.529,171.552,47.359,159.268
C06929=1027.092,337.427,-135.493,171.545,47.358,159.267
C06930=1027.085,337.179,-135.457,171.539,47.359,159.267
C06931=1027.078,336.960,-135.425,171.534,47.358,159.266
C06932=1027.071,336.741,-135.393,171.529,47.359,159.265
C06933=1027.065,336.522,-135.361,171.523,47.359,159.265
C06934=1027.058,336.303,-135.329,171.519,47.359,159.264
C06935=1027.052,336.085,-135.298,171.513,47.359,159.263
C06936=1027.045,335.865,-135.265,171.507,47.359,159.263
C06937=1027.039,335.646,-135.233,171.503,47.359,159.262
C06938=1027.032,335.428,-135.201,171.497,47.359,159.261
C06939=1027.025,335.180,-135.166,171.491,47.359,159.260
C06940=1027.017,334.933,-135.130,171.485,47.359,159.260
C06941=1027.010,334.685,-135.093,171.480,47.359,159.259
C06942=1027.003,334.438,-135.057,171.473,47.359,159.258
C06943=1026.996,334.191,-135.021,171.467,47.359,159.257
C06944=1026.989,333.943,-134.986,171.461,47.359,159.257
C06945=1026.981,333.696,-134.950,171.456,47.359,159.256
C06946=1026.974,333.449,-134.914,171.450,47.360,159.255
C06947=1026.966,333.202,-134.879,171.443,47.360,159.255
C06948=1026.958,332.954,-134.843,171.438,47.360,159.254
C06949=1026.952,332.707,-134.807,171.432,47.360,159.253
C06950=1026.944,332.459,-134.771,171.426,47.361,159.252
C06951=1026.937,332.213,-134.735,171.421,47.361,159.252
C06952=1026.929,331.964,-134.700,171.415,47.361,159.251
C06953=1026.922,331.718,-134.665,171.408,47.361,159.250
C06954=1026.914,331.470,-134.629,171.403,47.361,159.250
C06955=1026.907,331.223,-134.594,171.397,47.362,159.249
C06956=1026.900,330.975,-134.558,171.391,47.362,159.248
C06957=1026.893,330.728,-134.523,171.386,47.362,159.248
C06958=1026.885,330.480,-134.486,171.380,47.362,159.247
C06959=1026.878,330.233,-134.452,171.374,47.362,159.246
C06960=1026.871,329.986,-134.417,171.368,47.363,159.246
C06961=1026.863,329.738,-134.381,171.362,47.364,159.245
C06962=1026.857,329.491,-134.345,171.357,47.364,159.244
C06963=1026.849,329.243,-134.310,171.351,47.364,159.243
C06964=1026.842,328.996,-134.274,171.345,47.364,159.243
C06965=1026.835,328.749,-134.240,171.340,47.364,159.242
C06966=1026.827,328.501,-134.204,171.334,47.365,159.242
C06967=1026.821,328.254,-134.169,171.329,47.365,159.241
C06968=1026.813,328.007,-134.133,171.323,47.365,159.240
C06969=1026.806,327.759,-134.098,171.317,47.366,159.239
C06970=1026.799,327.512,-134.063,171.312,47.366,159.239
C06971=1026.792,327.265,-134.028,171.305,47.367,159.238
C06972=1026.784,327.017,-133.993,171.300,47.367,159.237
C06973=1026.777,326.769,-133.958,171.294,47.368,159.237
C06974=1026.769,326.522,-133.923,171.289,47.368,159.236
C06975=1026.762,326.274,-133.888,171.283,47.369,159.236
C06976=1026.755,326.027,-133.853,171.278,47.369,159.235
C06977=1026.747,325.780,-133.819,171.272,47.370,159.235
C06978=1026.740,325.532,-133.784,171.267,47.370,159.234
C06979=1026.732,325.284,-133.749,171.261,47.371,159.233
C06980=1026.725,325.037,-133.715,171.255,47.371,159.233
C06981=1026.718,324.790,-133.680,171.249,47.372,159.232
C06982=1026.710,324.542,-133.645,171.244,47.373,159.232
C06983=1026.704,324.294,-133.610,171.238,47.373,159.231
C06984=1026.696,324.047,-133.576,171.233,47.374,159.230
C06985=1026.689,323.800,-133.541,171.227,47.374,159.230
C06986=1026.682,323.553,-133.506,171.222,47.375,159.229
C06987=1026.674,323.304,-133.472,171.216,47.375,159.229
C06988=1026.667,323.057,-133.437,171.211,47.375,159.228
C06989=1026.660,322.810,-133.402,171.205,47.376,159.227
C06990=1026.653,322.562,-133.368,171.200,47.377,159.227
C06991=1026.646,322.341,-133.337,171.194,47.377,159.226
C06992=1026.640,322.120,-133.306,171.190,47.378,159.226
C06993=1026.634,321.899,-133.275,171.185,47.378,159.225
C06994=1026.627,321.677,-133.245,171.180,47.379,159.225
C06995=1026.620,321.457,-133.214,171.175,47.380,159.224
C06996=1026.614,321.235,-133.183,171.171,47.380,159.224
C06997=1026.608,321.014,-133.152,171.165,47.381,159.223
C06998=1026.601,320.793,-133.121,171.161,47.382,159.223
C06999=1026.594,320.545,-133.087,171.155,47.382,159.222
C07000=1026.587,320.298,-133.053,171.150,47.383,159.222
C07001=1026.580,320.050,-133.018,171.145,47.383,159.221
C07002=1026.573,319.803,-132.984,171.139,47.384,159.221
C07003=1026.565,319.556,-132.949,171.134,47.385,159.220
C07004=1026.559,319.308,-132.915,171.128,47.385,159.219
C07005=1026.551,319.061,-132.880,171.123,47.386,159.219
C07006=1026.545,318.813,-132.846,171.118,47.387,159.218
C07007=1026.538,318.565,-132.812,171.112,47.387,159.218
C07008=1026.530,318.318,-132.778,171.107,47.388,159.217
C07009=1026.524,318.070,-132.743,171.102,47.389,159.217
C07010=1026.516,317.822,-132.709,171.096,47.390,159.216
C07011=1026.509,317.575,-132.675,171.091,47.391,159.216
C07012=1026.502,317.327,-132.640,171.085,47.391,159.215
C07013=1026.495,317.080,-132.607,171.081,47.392,159.215
C07014=1026.488,316.833,-132.572,171.076,47.393,159.214
C07015=1026.482,316.585,-132.538,171.070,47.393,159.214
C07016=1026.475,316.338,-132.504,171.065,47.394,159.213
C07017=1026.467,316.090,-132.470,171.060,47.395,159.213
C07018=1026.461,315.842,-132.436,171.054,47.396,159.212
C07019=1026.453,315.595,-132.401,171.049,47.396,159.212
C07020=1026.446,315.347,-132.368,171.044,47.397,159.211
C07021=1026.440,315.100,-132.334,171.038,47.398,159.211
C07022=1026.433,314.852,-132.300,171.033,47.399,159.210
C07023=1026.426,314.605,-132.266,171.028,47.400,159.210
C07024=1026.419,314.357,-132.232,171.023,47.400,159.209
C07025=1026.412,314.109,-132.198,171.018,47.401,159.209
C07026=1026.406,313.862,-132.164,171.013,47.402,159.208
C07027=1026.398,313.615,-132.130,171.007,47.402,159.208
C07028=1026.392,313.367,-132.095,171.002,47.404,159.207
C07029=1026.385,313.119,-132.061,170.997,47.405,159.207
C07030=1026.378,312.872,-132.028,170.991,47.405,159.206
C07031=1026.372,312.624,-131.994,170.987,47.406,159.206
C07032=1026.364,312.377,-131.960,170.982,47.407,159.205
C07033=1026.358,312.130,-131.926,170.976,47.407,159.205
C07034=1026.351,311.882,-131.892,170.971,47.409,159.204
C07035=1026.344,311.633,-131.859,170.966,47.410,159.204
C07036=1026.338,311.386,-131.825,170.961,47.410,159.203
C07037=1026.331,311.139,-131.791,170.955,47.411,159.203
C07038=1026.324,310.891,-131.757,170.951,47.412,159.203
C07039=1026.317,310.644,-131.724,170.946,47.413,159.202
C07040=1026.310,310.396,-131.690,170.941,47.414,159.201
C07041=1026.303,310.148,-131.657,170.935,47.415,159.201
C07042=1026.296,309.901,-131.624,170.930,47.417,159.201
C07043=1026.289,309.653,-131.591,170.925,47.418,159.200
C07044=1026.281,309.405,-131.557,170.920,47.419,159.200
C07045=1026.275,309.158,-131.524,170.915,47.420,159.199
C07046=1026.268,308.910,-131.491,170.911,47.421,159.199
C07047=1026.260,308.663,-131.458,170.905,47.422,159.199
C07048=1026.254,308.415,-131.425,170.900,47.423,159.198
C07049=1026.246,308.168,-131.391,170.895,47.424,159.198
C07050=1026.239,307.920,-131.359,170.890,47.425,159.197
C07051=1026.233,307.701,-131.329,170.886,47.426,159.197
C07052=1026.227,307.482,-131.300,170.880,47.427,159.197
C07053=1026.220,307.264,-131.271,170.876,47.428,159.196
C07054=1026.215,307.045,-131.242,170.872,47.429,159.196
C07055=1026.208,306.826,-131.212,170.868,47.431,159.196
C07056=1026.203,306.607,-131.183,170.863,47.431,159.195
C07057=1026.196,306.389,-131.154,170.859,47.432,159.195
C07058=1026.190,306.170,-131.125,170.855,47.434,159.195
C07059=1026.183,305.922,-131.092,170.850,47.434,159.194
C07060=1026.176,305.675,-131.059,170.845,47.436,159.194
C07061=1026.169,305.427,-131.026,170.840,47.437,159.194
C07062=1026.162,305.180,-130.993,170.835,47.439,159.193
C07063=1026.155,304.932,-130.960,170.830,47.439,159.193
C07064=1026.148,304.684,-130.928,170.825,47.440,159.192
C07065=1026.141,304.436,-130.895,170.820,47.442,159.192
C07066=1026.135,304.189,-130.861,170.815,47.443,159.192
C07067=1026.127,303.941,-130.829,170.810,47.444,159.191
C07068=1026.121,303.693,-130.796,170.805,47.445,159.191
C07069=1026.114,303.445,-130.763,170.801,47.447,159.191
C07070=1026.107,303.198,-130.731,170.796,47.448,159.190
C07071=1026.100,302.951,-130.697,170.791,47.449,159.190
C07072=1026.093,302.703,-130.664,170.785,47.451,159.190
C07073=1026.086,302.455,-130.632,170.780,47.452,159.189
C07074=1026.079,302.207,-130.599,170.776,47.453,159.189
C07075=1026.073,301.959,-130.566,170.771,47.454,159.189
C07076=1026.066,301.712,-130.534,170.766,47.456,159.188
C07077=1026.059,301.464,-130.501,170.761,47.457,159.188
C07078=1026.052,301.217,-130.469,170.757,47.458,159.188
C07079=1026.045,300.968,-130.435,170.752,47.460,159.187
C07080=1026.039,300.721,-130.403,170.747,47.461,159.187
C07081=1026.032,300.473,-130.371,170.742,47.462,159.187
C07082=1026.025,300.225,-130.337,170.738,47.463,159.186
C07083=1026.019,299.977,-130.305,170.733,47.465,159.186
C07084=1026.012,299.730,-130.273,170.728,47.466,159.186
C07085=1026.005,299.482,-130.239,170.723,47.468,159.185
C07086=1025.999,299.234,-130.207,170.719,47.469,159.185
C07087=1025.992,298.987,-130.175,170.714,47.470,159.185
C07088=1025.985,298.739,-130.142,170.709,47.472,159.184
C07089=1025.978,298.491,-130.109,170.703,47.473,159.184
C07090=1025.971,298.244,-130.077,170.699,47.474,159.184
C07091=1025.965,297.996,-130.045,170.694,47.476,159.183
C07092=1025.959,297.748,-130.012,170.689,47.477,159.183
C07093=1025.951,297.500,-129.979,170.685,47.478,159.183
C07094=1025.945,297.252,-129.947,170.680,47.480,159.182
C07095=1025.939,297.005,-129.914,170.675,47.481,159.182
C07096=1025.932,296.757,-129.882,170.670,47.482,159.182
C07097=1025.926,296.509,-129.850,170.666,47.484,159.181
C07098=1025.918,296.261,-129.817,170.661,47.485,159.181
C07099=1025.912,296.014,-129.784,170.656,47.486,159.181
C07100=1025.906,295.766,-129.752,170.652,47.488,159.181
C07101=1025.899,295.518,-129.720,170.647,47.490,159.180
C07102=1025.893,295.271,-129.687,170.642,47.491,159.180
C07103=1025.887,295.022,-129.655,170.638,47.492,159.180
C07104=1025.879,294.774,-129.623,170.633,47.493,159.179
C07105=1025.873,294.527,-129.590,170.628,47.495,159.179
C07106=1025.866,294.279,-129.559,170.624,47.497,159.179
C07107=1025.860,294.031,-129.526,170.619,47.498,159.179
C07108=1025.853,293.784,-129.495,170.614,47.499,159.178
C07109=1025.847,293.536,-129.462,170.610,47.501,159.178
C07110=1025.840,293.288,-129.430,170.606,47.503,159.178
C07111=1025.834,293.078,-129.403,170.602,47.504,159.178
C07112=1025.828,292.868,-129.376,170.598,47.505,159.177
C07113=1025.823,292.657,-129.349,170.594,47.507,159.177
C07114=1025.817,292.448,-129.321,170.590,47.508,159.177
C07115=1025.811,292.237,-129.294,170.586,47.509,159.177
C07116=1025.805,292.028,-129.268,170.582,47.511,159.176
C07117=1025.800,291.817,-129.241,170.578,47.512,159.176
C07118=1025.794,291.608,-129.213,170.574,47.514,159.176
C07119=1025.787,291.360,-129.182,170.569,47.515,159.176
C07120=1025.781,291.112,-129.150,170.565,47.517,159.176
C07121=1025.774,290.864,-129.119,170.560,47.518,159.175
C07122=1025.767,290.617,-129.087,170.556,47.520,159.175
C07123=1025.760,290.369,-129.055,170.552,47.521,159.175
C07124=1025.754,290.121,-129.023,170.547,47.523,159.175
C07125=1025.747,289.872,-128.992,170.542,47.525,159.174
C07126=1025.740,289.625,-128.959,170.538,47.527,159.174
C07127=1025.733,289.377,-128.928,170.533,47.528,159.174
C07128=1025.726,289.129,-128.896,170.528,47.530,159.174
C07129=1025.720,288.881,-128.865,170.524,47.531,159.174
C07130=1025.714,288.633,-128.833,170.520,47.533,159.173
C07131=1025.707,288.385,-128.802,170.515,47.535,159.173
C07132=1025.700,288.137,-128.770,170.511,47.536,159.173
C07133=1025.694,287.889,-128.739,170.506,47.539,159.173
C07134=1025.687,287.641,-128.707,170.501,47.541,159.173
C07135=1025.680,287.393,-128.676,170.497,47.542,159.172
C07136=1025.673,287.145,-128.644,170.493,47.544,159.172
C07137=1025.667,286.897,-128.613,170.488,47.546,159.172
C07138=1025.661,286.650,-128.582,170.484,47.547,159.172
C07139=1025.654,286.402,-128.551,170.479,47.549,159.172
C07140=1025.647,286.154,-128.519,170.474,47.551,159.171
C07141=1025.641,285.906,-128.487,170.470,47.552,159.171
C07142=1025.634,285.658,-128.456,170.466,47.554,159.171
C07143=1025.628,285.410,-128.424,170.461,47.556,159.171
C07144=1025.620,285.163,-128.393,170.457,47.558,159.171
C07145=1025.614,284.915,-128.362,170.452,47.560,159.171
C07146=1025.607,284.667,-128.330,170.447,47.562,159.170
C07147=1025.600,284.418,-128.300,170.444,47.563,159.170
C07148=1025.594,284.171,-128.268,170.439,47.565,159.170
C07149=1025.587,283.923,-128.237,170.434,47.567,159.170
C07150=1025.580,283.675,-128.205,170.431,47.569,159.170
C07151=1025.574,283.427,-128.176,170.426,47.571,159.169
C07152=1025.567,283.179,-128.144,170.421,47.573,159.169
C07153=1025.560,282.931,-128.113,170.417,47.575,159.169
C07154=1025.554,282.683,-128.082,170.413,47.577,159.169
C07155=1025.547,282.435,-128.051,170.409,47.578,159.169
C07156=1025.540,282.187,-128.019,170.404,47.580,159.169
C07157=1025.533,281.939,-127.989,170.399,47.582,159.168
C07158=1025.527,281.692,-127.958,170.395,47.584,159.168
